// TIA Portal V20 export
// export: Created 2025-12-01T14:56:44.3017244Z, ExportSetting None, DisplayName Totally Integrated Automation Portal, DisplayVersion V20 Update 3, DisplayName TIA Portal Openness, DisplayVersion V20 Update 3, DisplayName TIA Portal Version Control Interface, DisplayVersion V20 Update 3, DisplayName STEP 7 Professional, DisplayVersion V20 Update 3, DisplayName STEP 7 Safety, DisplayVersion V20 Update 2, DisplayName WinCC Basic/Comfort/Advanced, DisplayVersion V20 Update 3, DisplayName WinCC Professional, DisplayVersion V20 Update 3, DisplayName WinCC Unified, DisplayVersion V20 Update 3
FUNCTION_BLOCK "FB246_M_STV_Carga_E1_S4"   // FB246, LAD
TITLE = Control del Ramal de Salidas
{ S7_Optimized_Access := 'FALSE' }
AUTHOR : VTD
NAME : 20160509
VERSION : 3.4
// stored: AutoNumber false, SetENOAutomatically false
   VAR_INPUT
      Mesa : UInt;   // Mesa de la FB
      Error_Tx : Bool;   // Error en el Tx
      EnTension : Bool;   // Existe Tension en la Mesa
      Termico_Tx : Bool;   // Proteccion del Tx E1E3
      pHsMx : Bool;   // pHs de la Mesa
      pHsMx_PR1 : Bool;   // pHs de Protrusion de la Mesa. Nota: No existe >> ON
      pHsMx_PR4 : Bool;   // pHs de Protrusion de la Mesa. Nota: No existe >> ON
      Avance_Tx : Bool;   // Avance del Tx
      Termico_TRx : Bool;   // Proteccion del TRx E2E4
      Pos_E2E4 : Bool;   // Pos. TR en E2E4
      Pos_E1E3 : Bool;   // Pos. TR en E1E3
      Avance_TRx : Bool;   // Avance del TRx E2E4
      EnMovimiento_TRx : Bool;   // En Movimiento la Elevacion del TRx
      LoadArrival : Bool;   // Load Arrival >>> VTD
      LoadComplete : Bool;   // LoadComplete >>> VTD
      MAnt_DescargaAct : Bool;   // E1 >> Mesa Anterior DescargaAct
      AVTF_MAnt_Mx : Bool;   // E1 >> Mesa Anterior AVTF
      P_Mens_Mant_Mx : Bool;   // E1 >> Mesa Anterior P_Mens
      PermisoPos_E2E4 : Bool;   // Permiso Pos. TR en E2E4
      PermisoPos_E1E3 : Bool;   // Permiso Pos. TR en E1E3
      Mx_PosReposo_E2E4 : Bool;   // Config >> Pos de Reposo Cargada
      Mx_TRElectrico : Bool;   // Config >> TR es Electrico
      Mx_TR_UP_E1E3 : Bool;   // Config >> TR Arriba en E1E3
      Mx_VelocidadLenta_In : Bool;   // Forzar a Velociada Lenta
      F_EnvMens_Mx : Bool;   // Fin de Envio de Mensaje
      OrdSal_S00 : Bool;   // Orden de Salida hacia el VTD
      V_CNT_pHsMx : Int := 1000;   // Valor de Presencia
      V_CNT_pHsMx_FTF : Int := 200;   // Valor para activar FTF. Nota: < = V_CNT_pHsMx.
      V_CNTSeg_pHsMx : Int := 2000;   // Valor de Seguriadad para Presencia
      V_CNT_PasoLenta : Int := 2000;   // Valor de Paso a Lenta
      V_CNT_ApHsMx : Int := 200;   // Valor de Ausencia
      V_CNTSeg_ApHsMx : Int := 2000;   // Valor de Seguriadad para Ausencia
      V_TOut_Tx_Mx : Int := 15000;   // TimeOut de Entrada por E1
      V_TOut_TR : Int := 5000;   // TimeOut de Elevacion del TR
      V_TOut_Interlock : Int := 5000;   // TimeOut de Fin del Interlock con el VTD
      V_TMP_Protrusion : Int := 200;   // TMP de Protrusion
      V_CNT_PerdidapHs : Int := 1000;   // CNT de Perdida de pHs
   END_VAR
   VAR_OUTPUT
      P_EnvMens_PMx : Bool;   // Permiso de Enviar Mensaje de Presencia
      P_EnvMens_AMx : Bool;   // Permiso de Enviar Mensaje de Ausencia
      P_RecepOK_Mx : Bool;   // Recepcion OK
      PTF_MAnt_Mx : Bool;   // E1 >> Mesa Anterior PTF
      FTF_MAnt_Mx : Bool;   // E1 >> Mesa Anterior FTF
   END_VAR
   VAR
      Anular_prE1 : Bool;   // ???
      Anular_prS4 : Bool;   // ???
      Mx_ET00 : Bool;
      Mx_ET01 : Bool;
      Mx_ET02 : Bool;
      Mx_ET08 : Bool;
      Mx_ET09 : Bool;
      Mx_ET10 : Bool;
      Mx_ET11 : Bool;
      Mx_ET12 : Bool;
      Mx_ET110 : Bool;
      Mx_ET111 : Bool;
      Mx_ET50 : Bool;
      Mx_ET51 : Bool;
      Mx_ET52 : Bool;
      Mx_ET150 : Bool;
      Mx_ET151 : Bool;
      Mx_ET152 : Bool;
      ProtocoloIniciado : Bool;   // Iniciado el Envio del Mensaje de Presencia
      CNT_pHsMx_FTF_OK : Bool;   // Enviar ya FTF
      STAT_EnvMens_PMx : Bool;   // Interna >> Envio del Mensaje de Presencia
      STAT_EnvMens_AMx : Bool;   // Interna >> Envio de Mensaje de Ausencia
      STAT_FTF_MAnt_Mx : Bool;   // Interna >> FTF de MAnt >> Mx
      CNT_pHsMx { S7_SetPoint := 'True'} : "FB910_CNT_UHS";   // CNT de la Presencia
      CNTSeg_pHsMx { S7_SetPoint := 'True'} : "FB910_CNT_UHS";   // CNT de Seguridad de la Presencia
      CNT_ApHsMx { S7_SetPoint := 'True'} : "FB910_CNT_UHS";   // CNT de la Ausencia
      CNTSeg_ApHsMx { S7_SetPoint := 'True'} : "FB910_CNT_UHS";   // CNT de Seguridad de la Ausencia
      TMP_EnTension { S7_SetPoint := 'True'} : "FB910_CNT_UHS";
      TOut_Av_Mx { S7_SetPoint := 'True'} : "FB910_CNT_UHS";   // Time Out de Entrada de E1
      TOut_Subir_TR { S7_SetPoint := 'True'} : "FB910_CNT_UHS";   // Time Out de Subida del TR
      TOut_Bajar_TR { S7_SetPoint := 'True'} : "FB910_CNT_UHS";   // Time Out de Bajada del TR
      TOut_Interlock { S7_SetPoint := 'True'} : "FB910_CNT_UHS";   // Time Out de Fin de Interlock con el VTD
      TMP_Protrusion { S7_SetPoint := 'True'} : "FB910_CNT_UHS";   // TMP de la Protrusion
      CNT_PerdidapHs { S7_SetPoint := 'True'} : "FB910_CNT_UHS";   // CNT de Perdida de pHs
      Interlock_manual { S7_SetPoint := 'True'} : "UDT_Interlock_manual_STV";
   END_VAR
   VAR_TEMP
      EstadoZona : "EstadoZona";   // Estado de Zona de la Mesa
      EstadoVI : "EstadosMesa";   // Estado del Vehiculo Inteliguente de la Mesa
      ConfigFB : "UDT_ConfigFB";   // Configuracion de la FB de la Mesa
      Interlock : "UDT_Interlock_STV";
      V_Protrusion : Int;
      retval : Int;
      cero : USInt;
      Aux_ET00 : Bool;
   END_VAR
BEGIN

REGION Network 1: INICIALIZAR - Recoger las Variables de Estado de la Mesa
   // Se recoge - Estado_CBx
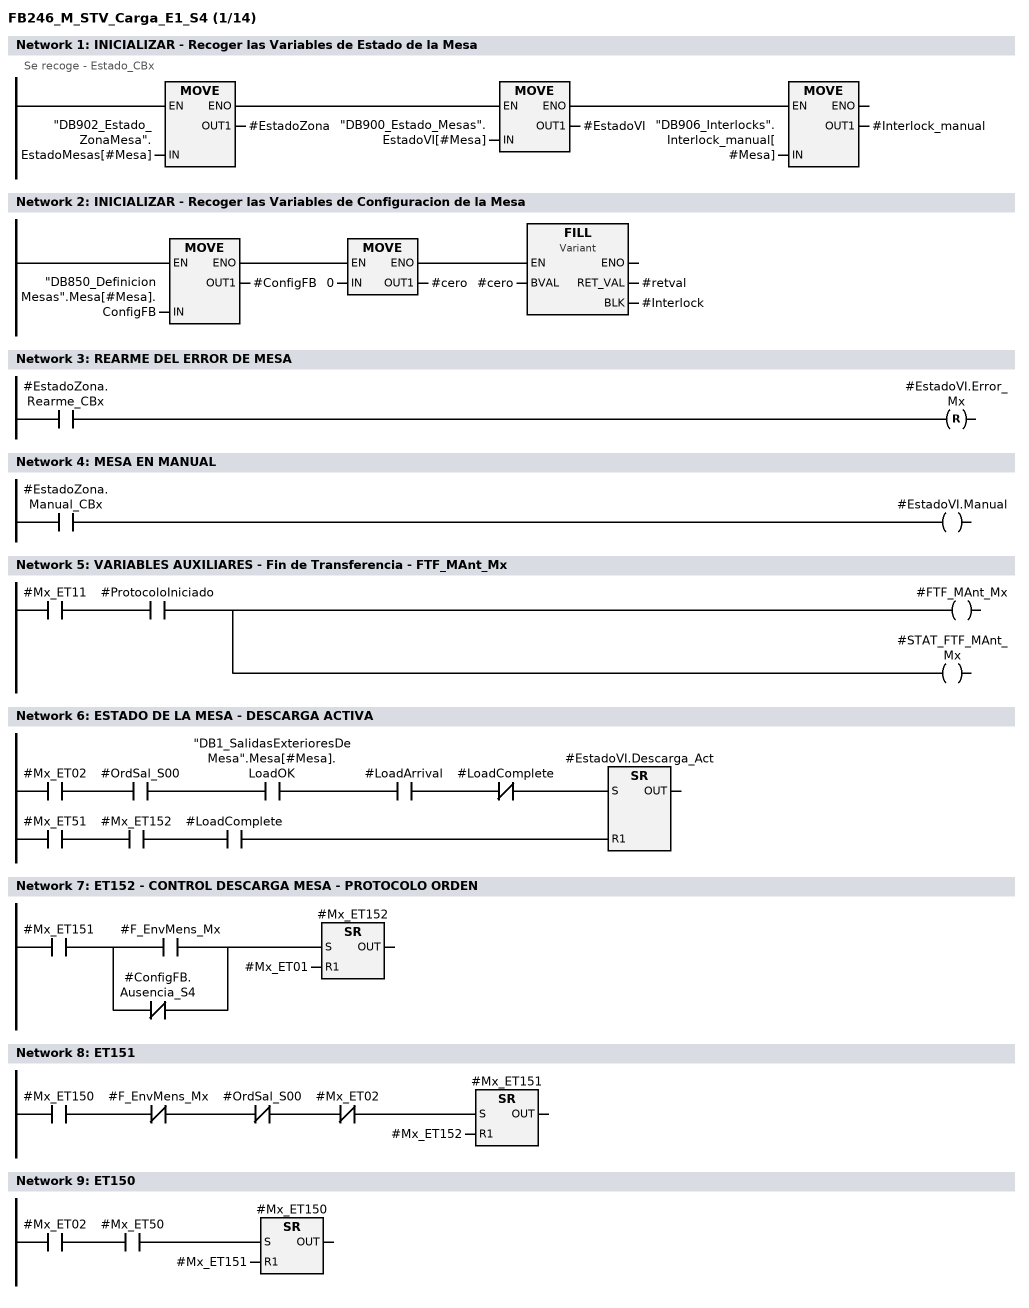
   RUNG wire#powerrail
      Move(in := "DB902_Estado_ZonaMesa".EstadoMesas[#Mesa], out1 => #EstadoZona)
      Move(in := "DB900_Estado_Mesas".EstadoVI[#Mesa], out1 => #EstadoVI)
      Move(in := "DB906_Interlocks".Interlock_manual[#Mesa], out1 => #Interlock_manual)
   END_RUNG
   // the same network as SCL:
   #EstadoZona := "DB902_Estado_ZonaMesa".EstadoMesas[#Mesa];
   #EstadoVI := "DB900_Estado_Mesas".EstadoVI[#Mesa];
   #Interlock_manual := "DB906_Interlocks".Interlock_manual[#Mesa];
END_REGION

REGION Network 2: INICIALIZAR - Recoger las Variables de Configuracion de la Mesa
   RUNG wire#powerrail
      Move(in := "DB850_DefinicionMesas".Mesa[#Mesa].ConfigFB, out1 => #ConfigFB)
      Move(in := 0, out1 => #cero)
      { S7_Templates := "ptr_type := Variant" } FILL(BVAL := #cero, RET_VAL => #retval, BLK => #Interlock)
   END_RUNG
   // the same network as SCL:
   #ConfigFB := "DB850_DefinicionMesas".Mesa[#Mesa].ConfigFB;
   #cero := 0;
   #retval := FILL(BVAL := #cero, BLK => #Interlock);
END_REGION

REGION Network 3: REARME DEL ERROR DE MESA
   RUNG wire#powerrail
      Contact( #EstadoZona.Rearme_CBx )
      R_Coil( #EstadoVI.Error_Mx )
   END_RUNG
   // the same network as SCL:
   IF #EstadoZona.Rearme_CBx THEN #EstadoVI.Error_Mx := FALSE; END_IF;
END_REGION

REGION Network 4: MESA EN MANUAL
   RUNG wire#powerrail
      Contact( #EstadoZona.Manual_CBx )
      Coil( #EstadoVI.Manual )
   END_RUNG
   // the same network as SCL:
   #EstadoVI.Manual := #EstadoZona.Manual_CBx;
END_REGION

REGION Network 5: VARIABLES AUXILIARES - Fin de Transferencia - FTF_MAnt_Mx
   RUNG wire#powerrail
      Contact( #Mx_ET11 )
      Contact( #ProtocoloIniciado )
      wire#w1
      Coil( #FTF_MAnt_Mx )
   END_RUNG
   RUNG wire#w1
      Coil( #STAT_FTF_MAnt_Mx )
   END_RUNG
   // the same network as SCL:
   #FTF_MAnt_Mx := #Mx_ET11 AND #ProtocoloIniciado;
   #STAT_FTF_MAnt_Mx := #FTF_MAnt_Mx;
END_REGION

REGION Network 6: ESTADO DE LA MESA - DESCARGA ACTIVA
   RUNG wire#powerrail
      Contact( #Mx_ET02 )
      Contact( #OrdSal_S00 )
      Contact( "DB1_SalidasExterioresDeMesa".Mesa[#Mesa].LoadOK )
      Contact( #LoadArrival )
      I_Contact( #LoadComplete )
      S_SR(operand := #EstadoVI.Descarga_Act, r1 := wire#w1)
   END_RUNG
   RUNG wire#powerrail
      Contact( #Mx_ET51 )
      Contact( #Mx_ET152 )
      Contact( #LoadComplete )
   END_RUNG wire#w1
   // the same network as SCL:
   IF #Mx_ET02 AND #OrdSal_S00 AND "DB1_SalidasExterioresDeMesa".Mesa[#Mesa].LoadOK AND #LoadArrival AND NOT #LoadComplete THEN
       #EstadoVI.Descarga_Act := TRUE;   // SR flip-flop
   END_IF;
   IF #Mx_ET51 AND #Mx_ET152 AND #LoadComplete THEN #EstadoVI.Descarga_Act := FALSE; END_IF;
END_REGION

REGION Network 7: ET152 - CONTROL DESCARGA MESA - PROTOCOLO ORDEN
   RUNG wire#powerrail
      Contact( #Mx_ET151 )
      wire#w1
      Contact( #F_EnvMens_Mx )
      wire#w2
      S_SR(operand := #Mx_ET152, r1 := #Mx_ET01)
   END_RUNG
   RUNG wire#w1
      I_Contact( #ConfigFB.Ausencia_S4 )
   END_RUNG wire#w2
   // the same network as SCL:
   IF #Mx_ET151 AND (#F_EnvMens_Mx OR NOT #ConfigFB.Ausencia_S4) THEN
       #Mx_ET152 := TRUE;   // SR flip-flop
   END_IF;
   IF #Mx_ET01 THEN #Mx_ET152 := FALSE; END_IF;
END_REGION

REGION Network 8: ET151
   RUNG wire#powerrail
      Contact( #Mx_ET150 )
      I_Contact( #F_EnvMens_Mx )
      I_Contact( #OrdSal_S00 )
      I_Contact( #Mx_ET02 )
      S_SR(operand := #Mx_ET151, r1 := #Mx_ET152)
   END_RUNG
   // the same network as SCL:
   IF #Mx_ET150 AND NOT #F_EnvMens_Mx AND NOT #OrdSal_S00 AND NOT #Mx_ET02 THEN
       #Mx_ET151 := TRUE;   // SR flip-flop
   END_IF;
   IF #Mx_ET152 THEN #Mx_ET151 := FALSE; END_IF;
END_REGION

REGION Network 9: ET150
   RUNG wire#powerrail
      Contact( #Mx_ET02 )
      Contact( #Mx_ET50 )
      S_SR(operand := #Mx_ET150, r1 := #Mx_ET151)
   END_RUNG
   // the same network as SCL:
   IF #Mx_ET02 AND #Mx_ET50 THEN
       #Mx_ET150 := TRUE;   // SR flip-flop
   END_IF;
   IF #Mx_ET151 THEN #Mx_ET150 := FALSE; END_IF;
END_REGION

REGION Network 10: ET52 - CONTROL DESCARGA MESA
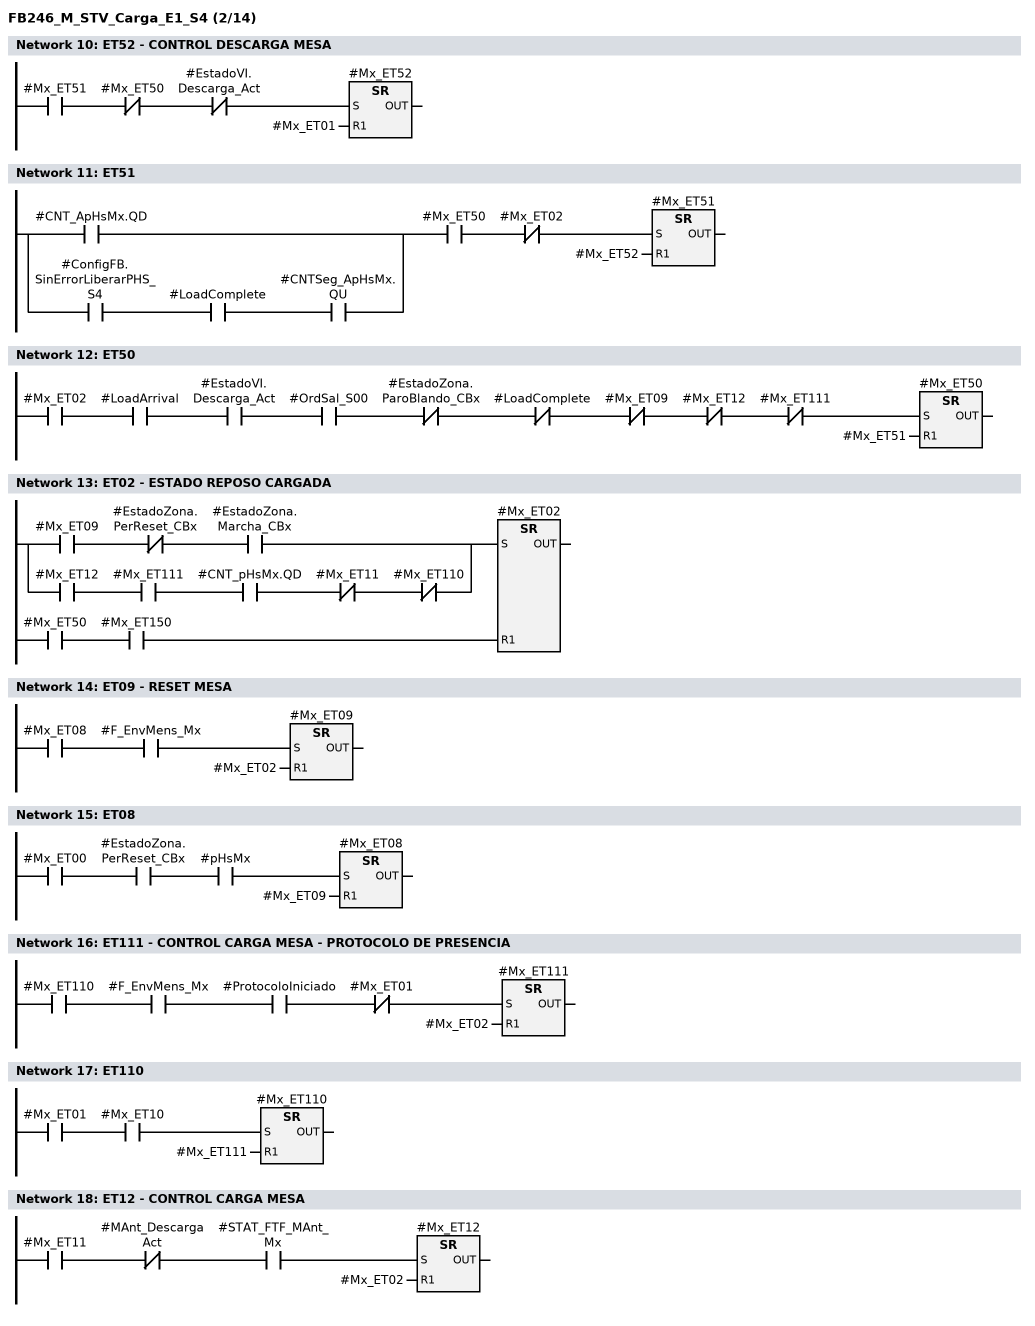
   RUNG wire#powerrail
      Contact( #Mx_ET51 )
      I_Contact( #Mx_ET50 )
      I_Contact( #EstadoVI.Descarga_Act )
      S_SR(operand := #Mx_ET52, r1 := #Mx_ET01)
   END_RUNG
   // the same network as SCL:
   IF #Mx_ET51 AND NOT #Mx_ET50 AND NOT #EstadoVI.Descarga_Act THEN
       #Mx_ET52 := TRUE;   // SR flip-flop
   END_IF;
   IF #Mx_ET01 THEN #Mx_ET52 := FALSE; END_IF;
END_REGION

REGION Network 11: ET51
   RUNG wire#powerrail
      Contact( #CNT_ApHsMx.QD )
      wire#w1
      Contact( #Mx_ET50 )
      I_Contact( #Mx_ET02 )
      S_SR(operand := #Mx_ET51, r1 := #Mx_ET52)
   END_RUNG
   RUNG wire#powerrail
      Contact( #ConfigFB.SinErrorLiberarPHS_S4 )
      Contact( #LoadComplete )
      Contact( #CNTSeg_ApHsMx.QU )
   END_RUNG wire#w1
   // the same network as SCL:
   IF (#CNT_ApHsMx.QD OR (#ConfigFB.SinErrorLiberarPHS_S4 AND #LoadComplete AND #CNTSeg_ApHsMx.QU)) AND #Mx_ET50 AND NOT #Mx_ET02 THEN
       #Mx_ET51 := TRUE;   // SR flip-flop
   END_IF;
   IF #Mx_ET52 THEN #Mx_ET51 := FALSE; END_IF;
END_REGION

REGION Network 12: ET50
   RUNG wire#powerrail
      Contact( #Mx_ET02 )
      Contact( #LoadArrival )
      Contact( #EstadoVI.Descarga_Act )
      Contact( #OrdSal_S00 )
      I_Contact( #EstadoZona.ParoBlando_CBx )
      I_Contact( #LoadComplete )
      I_Contact( #Mx_ET09 )
      I_Contact( #Mx_ET12 )
      I_Contact( #Mx_ET111 )
      S_SR(operand := #Mx_ET50, r1 := #Mx_ET51)
   END_RUNG
   // the same network as SCL:
   IF #Mx_ET02 AND #LoadArrival AND #EstadoVI.Descarga_Act AND #OrdSal_S00 AND NOT #EstadoZona.ParoBlando_CBx AND NOT #LoadComplete AND NOT #Mx_ET09 AND NOT #Mx_ET12 AND NOT #Mx_ET111 THEN
       #Mx_ET50 := TRUE;   // SR flip-flop
   END_IF;
   IF #Mx_ET51 THEN #Mx_ET50 := FALSE; END_IF;
END_REGION

REGION Network 13: ET02 - ESTADO REPOSO CARGADA
   RUNG wire#powerrail
      Contact( #Mx_ET09 )
      I_Contact( #EstadoZona.PerReset_CBx )
      Contact( #EstadoZona.Marcha_CBx )
      wire#w1
      S_SR(operand := #Mx_ET02, r1 := wire#w2)
   END_RUNG
   RUNG wire#powerrail
      Contact( #Mx_ET12 )
      Contact( #Mx_ET111 )
      Contact( #CNT_pHsMx.QD )
      I_Contact( #Mx_ET11 )
      I_Contact( #Mx_ET110 )
   END_RUNG wire#w1
   RUNG wire#powerrail
      Contact( #Mx_ET50 )
      Contact( #Mx_ET150 )
   END_RUNG wire#w2
   // the same network as SCL:
   IF (#Mx_ET09 AND NOT #EstadoZona.PerReset_CBx AND #EstadoZona.Marcha_CBx) OR (#Mx_ET12 AND #Mx_ET111 AND #CNT_pHsMx.QD AND NOT #Mx_ET11 AND NOT #Mx_ET110) THEN
       #Mx_ET02 := TRUE;   // SR flip-flop
   END_IF;
   IF #Mx_ET50 AND #Mx_ET150 THEN #Mx_ET02 := FALSE; END_IF;
END_REGION

REGION Network 14: ET09 - RESET MESA
   RUNG wire#powerrail
      Contact( #Mx_ET08 )
      Contact( #F_EnvMens_Mx )
      S_SR(operand := #Mx_ET09, r1 := #Mx_ET02)
   END_RUNG
   // the same network as SCL:
   IF #Mx_ET08 AND #F_EnvMens_Mx THEN
       #Mx_ET09 := TRUE;   // SR flip-flop
   END_IF;
   IF #Mx_ET02 THEN #Mx_ET09 := FALSE; END_IF;
END_REGION

REGION Network 15: ET08
   RUNG wire#powerrail
      Contact( #Mx_ET00 )
      Contact( #EstadoZona.PerReset_CBx )
      Contact( #pHsMx )
      S_SR(operand := #Mx_ET08, r1 := #Mx_ET09)
   END_RUNG
   // the same network as SCL:
   IF #Mx_ET00 AND #EstadoZona.PerReset_CBx AND #pHsMx THEN
       #Mx_ET08 := TRUE;   // SR flip-flop
   END_IF;
   IF #Mx_ET09 THEN #Mx_ET08 := FALSE; END_IF;
END_REGION

REGION Network 16: ET111 - CONTROL CARGA MESA - PROTOCOLO DE PRESENCIA
   RUNG wire#powerrail
      Contact( #Mx_ET110 )
      Contact( #F_EnvMens_Mx )
      Contact( #ProtocoloIniciado )
      I_Contact( #Mx_ET01 )
      S_SR(operand := #Mx_ET111, r1 := #Mx_ET02)
   END_RUNG
   // the same network as SCL:
   IF #Mx_ET110 AND #F_EnvMens_Mx AND #ProtocoloIniciado AND NOT #Mx_ET01 THEN
       #Mx_ET111 := TRUE;   // SR flip-flop
   END_IF;
   IF #Mx_ET02 THEN #Mx_ET111 := FALSE; END_IF;
END_REGION

REGION Network 17: ET110
   RUNG wire#powerrail
      Contact( #Mx_ET01 )
      Contact( #Mx_ET10 )
      S_SR(operand := #Mx_ET110, r1 := #Mx_ET111)
   END_RUNG
   // the same network as SCL:
   IF #Mx_ET01 AND #Mx_ET10 THEN
       #Mx_ET110 := TRUE;   // SR flip-flop
   END_IF;
   IF #Mx_ET111 THEN #Mx_ET110 := FALSE; END_IF;
END_REGION

REGION Network 18: ET12 - CONTROL CARGA MESA
   RUNG wire#powerrail
      Contact( #Mx_ET11 )
      I_Contact( #MAnt_DescargaAct )
      Contact( #STAT_FTF_MAnt_Mx )
      S_SR(operand := #Mx_ET12, r1 := #Mx_ET02)
   END_RUNG
   // the same network as SCL:
   IF #Mx_ET11 AND NOT #MAnt_DescargaAct AND #STAT_FTF_MAnt_Mx THEN
       #Mx_ET12 := TRUE;   // SR flip-flop
   END_IF;
   IF #Mx_ET02 THEN #Mx_ET12 := FALSE; END_IF;
END_REGION

REGION Network 19: ET11
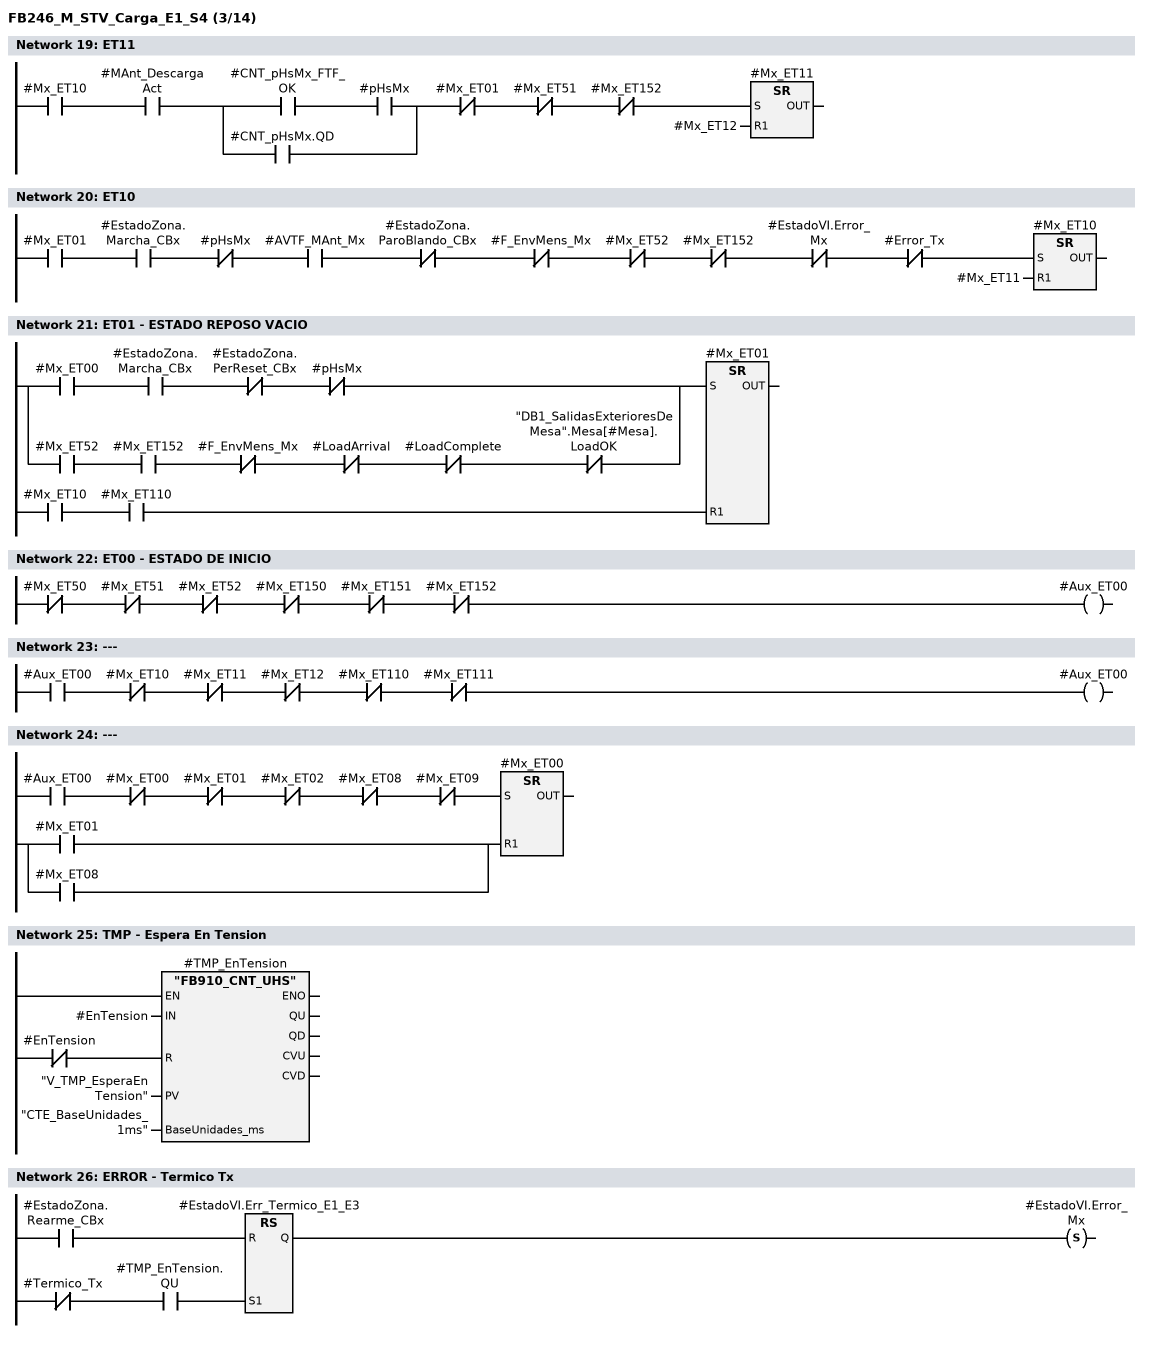
   RUNG wire#powerrail
      Contact( #Mx_ET10 )
      Contact( #MAnt_DescargaAct )
      wire#w1
      Contact( #CNT_pHsMx_FTF_OK )
      Contact( #pHsMx )
      wire#w2
      I_Contact( #Mx_ET01 )
      I_Contact( #Mx_ET51 )
      I_Contact( #Mx_ET152 )
      S_SR(operand := #Mx_ET11, r1 := #Mx_ET12)
   END_RUNG
   RUNG wire#w1
      Contact( #CNT_pHsMx.QD )
   END_RUNG wire#w2
   // the same network as SCL:
   IF #Mx_ET10 AND #MAnt_DescargaAct AND ((#CNT_pHsMx_FTF_OK AND #pHsMx) OR #CNT_pHsMx.QD) AND NOT #Mx_ET01 AND NOT #Mx_ET51 AND NOT #Mx_ET152 THEN
       #Mx_ET11 := TRUE;   // SR flip-flop
   END_IF;
   IF #Mx_ET12 THEN #Mx_ET11 := FALSE; END_IF;
END_REGION

REGION Network 20: ET10
   RUNG wire#powerrail
      Contact( #Mx_ET01 )
      Contact( #EstadoZona.Marcha_CBx )
      I_Contact( #pHsMx )
      Contact( #AVTF_MAnt_Mx )
      I_Contact( #EstadoZona.ParoBlando_CBx )
      I_Contact( #F_EnvMens_Mx )
      I_Contact( #Mx_ET52 )
      I_Contact( #Mx_ET152 )
      I_Contact( #EstadoVI.Error_Mx )
      I_Contact( #Error_Tx )
      S_SR(operand := #Mx_ET10, r1 := #Mx_ET11)
   END_RUNG
   // the same network as SCL:
   IF #Mx_ET01 AND #EstadoZona.Marcha_CBx AND NOT #pHsMx AND #AVTF_MAnt_Mx AND NOT #EstadoZona.ParoBlando_CBx AND NOT #F_EnvMens_Mx AND NOT #Mx_ET52 AND NOT #Mx_ET152 AND NOT #EstadoVI.Error_Mx AND NOT #Error_Tx THEN
       #Mx_ET10 := TRUE;   // SR flip-flop
   END_IF;
   IF #Mx_ET11 THEN #Mx_ET10 := FALSE; END_IF;
END_REGION

REGION Network 21: ET01 - ESTADO REPOSO VACIO
   RUNG wire#powerrail
      Contact( #Mx_ET00 )
      Contact( #EstadoZona.Marcha_CBx )
      I_Contact( #EstadoZona.PerReset_CBx )
      I_Contact( #pHsMx )
      wire#w1
      S_SR(operand := #Mx_ET01, r1 := wire#w2)
   END_RUNG
   RUNG wire#powerrail
      Contact( #Mx_ET52 )
      Contact( #Mx_ET152 )
      I_Contact( #F_EnvMens_Mx )
      I_Contact( #LoadArrival )
      I_Contact( #LoadComplete )
      I_Contact( "DB1_SalidasExterioresDeMesa".Mesa[#Mesa].LoadOK )
   END_RUNG wire#w1
   RUNG wire#powerrail
      Contact( #Mx_ET10 )
      Contact( #Mx_ET110 )
   END_RUNG wire#w2
   // the same network as SCL:
   IF (#Mx_ET00 AND #EstadoZona.Marcha_CBx AND NOT #EstadoZona.PerReset_CBx AND NOT #pHsMx) OR (#Mx_ET52 AND #Mx_ET152 AND NOT #F_EnvMens_Mx AND NOT #LoadArrival AND NOT #LoadComplete AND NOT "DB1_SalidasExterioresDeMesa".Mesa[#Mesa].LoadOK) THEN
       #Mx_ET01 := TRUE;   // SR flip-flop
   END_IF;
   IF #Mx_ET10 AND #Mx_ET110 THEN #Mx_ET01 := FALSE; END_IF;
END_REGION

REGION Network 22: ET00 - ESTADO DE INICIO
   RUNG wire#powerrail
      I_Contact( #Mx_ET50 )
      I_Contact( #Mx_ET51 )
      I_Contact( #Mx_ET52 )
      I_Contact( #Mx_ET150 )
      I_Contact( #Mx_ET151 )
      I_Contact( #Mx_ET152 )
      Coil( #Aux_ET00 )
   END_RUNG
   // the same network as SCL:
   #Aux_ET00 := NOT #Mx_ET50 AND NOT #Mx_ET51 AND NOT #Mx_ET52 AND NOT #Mx_ET150 AND NOT #Mx_ET151 AND NOT #Mx_ET152;
END_REGION

REGION Network 23: ---
   RUNG wire#powerrail
      Contact( #Aux_ET00 )
      I_Contact( #Mx_ET10 )
      I_Contact( #Mx_ET11 )
      I_Contact( #Mx_ET12 )
      I_Contact( #Mx_ET110 )
      I_Contact( #Mx_ET111 )
      Coil( #Aux_ET00 )
   END_RUNG
   // the same network as SCL:
   #Aux_ET00 := #Aux_ET00 AND NOT #Mx_ET10 AND NOT #Mx_ET11 AND NOT #Mx_ET12 AND NOT #Mx_ET110 AND NOT #Mx_ET111;
END_REGION

REGION Network 24: ---
   RUNG wire#powerrail
      Contact( #Aux_ET00 )
      I_Contact( #Mx_ET00 )
      I_Contact( #Mx_ET01 )
      I_Contact( #Mx_ET02 )
      I_Contact( #Mx_ET08 )
      I_Contact( #Mx_ET09 )
      S_SR(operand := #Mx_ET00, r1 := wire#w1)
   END_RUNG
   RUNG wire#powerrail
      Contact( #Mx_ET01 )
   END_RUNG wire#w1
   RUNG wire#powerrail
      Contact( #Mx_ET08 )
   END_RUNG wire#w1
   // the same network as SCL:
   IF #Aux_ET00 AND NOT #Mx_ET00 AND NOT #Mx_ET01 AND NOT #Mx_ET02 AND NOT #Mx_ET08 AND NOT #Mx_ET09 THEN
       #Mx_ET00 := TRUE;   // SR flip-flop
   END_IF;
   IF #Mx_ET01 OR #Mx_ET08 THEN #Mx_ET00 := FALSE; END_IF;
END_REGION

REGION Network 25: TMP - Espera En Tension
   RUNG wire#powerrail
      #TMP_EnTension(R := wire#w1, IN := #EnTension, PV := "V_TMP_EsperaEnTension", BaseUnidades_ms := "CTE_BaseUnidades_1ms", QU =>, QD =>, CVU =>, CVD =>)
   END_RUNG
   RUNG wire#powerrail
      I_Contact( #EnTension )
   END_RUNG wire#w1
   // the same network as SCL:
   #TMP_EnTension(IN := #EnTension,   // "FB910_CNT_UHS"
                  R := NOT #EnTension,
                  PV := "V_TMP_EsperaEnTension",
                  BaseUnidades_ms := "CTE_BaseUnidades_1ms");
END_REGION

REGION Network 26: ERROR - Termico Tx
   RUNG wire#powerrail
      Contact( #EstadoZona.Rearme_CBx )
      S_RS(operand := #EstadoVI.Err_Termico_E1_E3, s1 := wire#w1)
      S_Coil( #EstadoVI.Error_Mx )
   END_RUNG
   RUNG wire#powerrail
      I_Contact( #Termico_Tx )
      Contact( #TMP_EnTension.QU )
   END_RUNG wire#w1
   // the same network as SCL:
   IF #EstadoZona.Rearme_CBx THEN
       #EstadoVI.Err_Termico_E1_E3 := FALSE;   // RS flip-flop
   END_IF;
   IF NOT #Termico_Tx AND #TMP_EnTension.QU THEN #EstadoVI.Err_Termico_E1_E3 := TRUE; END_IF;
   IF #EstadoVI.Err_Termico_E1_E3 THEN #EstadoVI.Error_Mx := TRUE; END_IF;
END_REGION

REGION Network 27: ERROR - Termico TRx
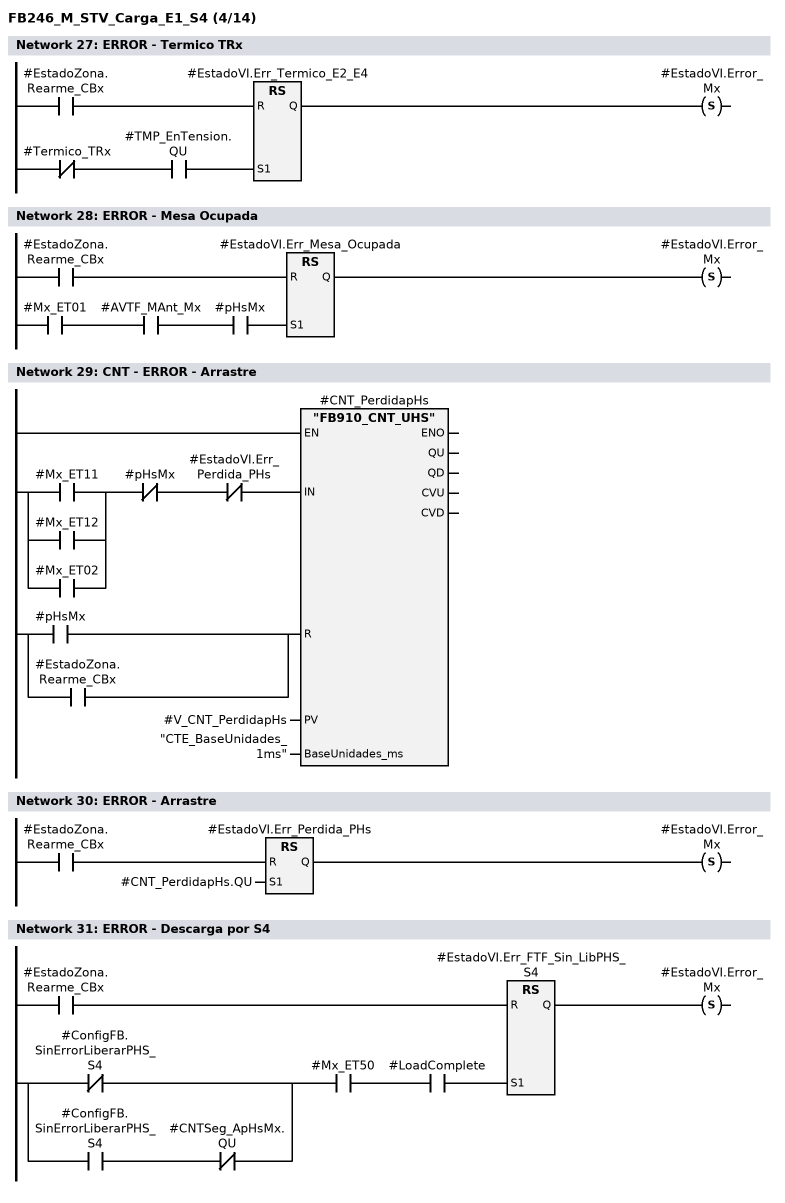
   RUNG wire#powerrail
      Contact( #EstadoZona.Rearme_CBx )
      S_RS(operand := #EstadoVI.Err_Termico_E2_E4, s1 := wire#w1)
      S_Coil( #EstadoVI.Error_Mx )
   END_RUNG
   RUNG wire#powerrail
      I_Contact( #Termico_TRx )
      Contact( #TMP_EnTension.QU )
   END_RUNG wire#w1
   // the same network as SCL:
   IF #EstadoZona.Rearme_CBx THEN
       #EstadoVI.Err_Termico_E2_E4 := FALSE;   // RS flip-flop
   END_IF;
   IF NOT #Termico_TRx AND #TMP_EnTension.QU THEN #EstadoVI.Err_Termico_E2_E4 := TRUE; END_IF;
   IF #EstadoVI.Err_Termico_E2_E4 THEN #EstadoVI.Error_Mx := TRUE; END_IF;
END_REGION

REGION Network 28: ERROR - Mesa Ocupada
   RUNG wire#powerrail
      Contact( #EstadoZona.Rearme_CBx )
      S_RS(operand := #EstadoVI.Err_Mesa_Ocupada, s1 := wire#w1)
      S_Coil( #EstadoVI.Error_Mx )
   END_RUNG
   RUNG wire#powerrail
      Contact( #Mx_ET01 )
      Contact( #AVTF_MAnt_Mx )
      Contact( #pHsMx )
   END_RUNG wire#w1
   // the same network as SCL:
   IF #EstadoZona.Rearme_CBx THEN
       #EstadoVI.Err_Mesa_Ocupada := FALSE;   // RS flip-flop
   END_IF;
   IF #Mx_ET01 AND #AVTF_MAnt_Mx AND #pHsMx THEN #EstadoVI.Err_Mesa_Ocupada := TRUE; END_IF;
   IF #EstadoVI.Err_Mesa_Ocupada THEN #EstadoVI.Error_Mx := TRUE; END_IF;
END_REGION

REGION Network 29: CNT - ERROR - Arrastre
   RUNG wire#powerrail
      #CNT_PerdidapHs(IN := wire#w2, R := wire#w3, PV := #V_CNT_PerdidapHs, BaseUnidades_ms := "CTE_BaseUnidades_1ms", QU =>, QD =>, CVU =>, CVD =>)
   END_RUNG
   RUNG wire#powerrail
      Contact( #Mx_ET11 )
      wire#w1
      I_Contact( #pHsMx )
      I_Contact( #EstadoVI.Err_Perdida_PHs )
   END_RUNG wire#w2
   RUNG wire#powerrail
      Contact( #Mx_ET12 )
   END_RUNG wire#w1
   RUNG wire#powerrail
      Contact( #Mx_ET02 )
   END_RUNG wire#w1
   RUNG wire#powerrail
      Contact( #pHsMx )
   END_RUNG wire#w3
   RUNG wire#powerrail
      Contact( #EstadoZona.Rearme_CBx )
   END_RUNG wire#w3
   // the same network as SCL:
   #CNT_PerdidapHs(IN := (#Mx_ET11 OR #Mx_ET12 OR #Mx_ET02) AND NOT #pHsMx AND NOT #EstadoVI.Err_Perdida_PHs,   // "FB910_CNT_UHS"
                   R := #pHsMx OR #EstadoZona.Rearme_CBx,
                   PV := #V_CNT_PerdidapHs,
                   BaseUnidades_ms := "CTE_BaseUnidades_1ms");
END_REGION

REGION Network 30: ERROR - Arrastre
   RUNG wire#powerrail
      Contact( #EstadoZona.Rearme_CBx )
      S_RS(operand := #EstadoVI.Err_Perdida_PHs, s1 := #CNT_PerdidapHs.QU)
      S_Coil( #EstadoVI.Error_Mx )
   END_RUNG
   // the same network as SCL:
   IF #EstadoZona.Rearme_CBx THEN
       #EstadoVI.Err_Perdida_PHs := FALSE;   // RS flip-flop
   END_IF;
   IF #CNT_PerdidapHs.QU THEN #EstadoVI.Err_Perdida_PHs := TRUE; END_IF;
   IF #EstadoVI.Err_Perdida_PHs THEN #EstadoVI.Error_Mx := TRUE; END_IF;
END_REGION

REGION Network 31: ERROR - Descarga por S4
   RUNG wire#powerrail
      Contact( #EstadoZona.Rearme_CBx )
      S_RS(operand := #EstadoVI.Err_FTF_Sin_LibPHS_S4, s1 := wire#w2)
      S_Coil( #EstadoVI.Error_Mx )
   END_RUNG
   RUNG wire#powerrail
      I_Contact( #ConfigFB.SinErrorLiberarPHS_S4 )
      wire#w1
      Contact( #Mx_ET50 )
      Contact( #LoadComplete )
   END_RUNG wire#w2
   RUNG wire#powerrail
      Contact( #ConfigFB.SinErrorLiberarPHS_S4 )
      I_Contact( #CNTSeg_ApHsMx.QU )
   END_RUNG wire#w1
   // the same network as SCL:
   IF #EstadoZona.Rearme_CBx THEN
       #EstadoVI.Err_FTF_Sin_LibPHS_S4 := FALSE;   // RS flip-flop
   END_IF;
   IF (NOT #ConfigFB.SinErrorLiberarPHS_S4 OR (#ConfigFB.SinErrorLiberarPHS_S4 AND NOT #CNTSeg_ApHsMx.QU)) AND #Mx_ET50 AND #LoadComplete THEN
       #EstadoVI.Err_FTF_Sin_LibPHS_S4 := TRUE;
   END_IF;
   IF #EstadoVI.Err_FTF_Sin_LibPHS_S4 THEN #EstadoVI.Error_Mx := TRUE; END_IF;
END_REGION

REGION Network 32: TMP - ERROR - TimeOut Avance Tx
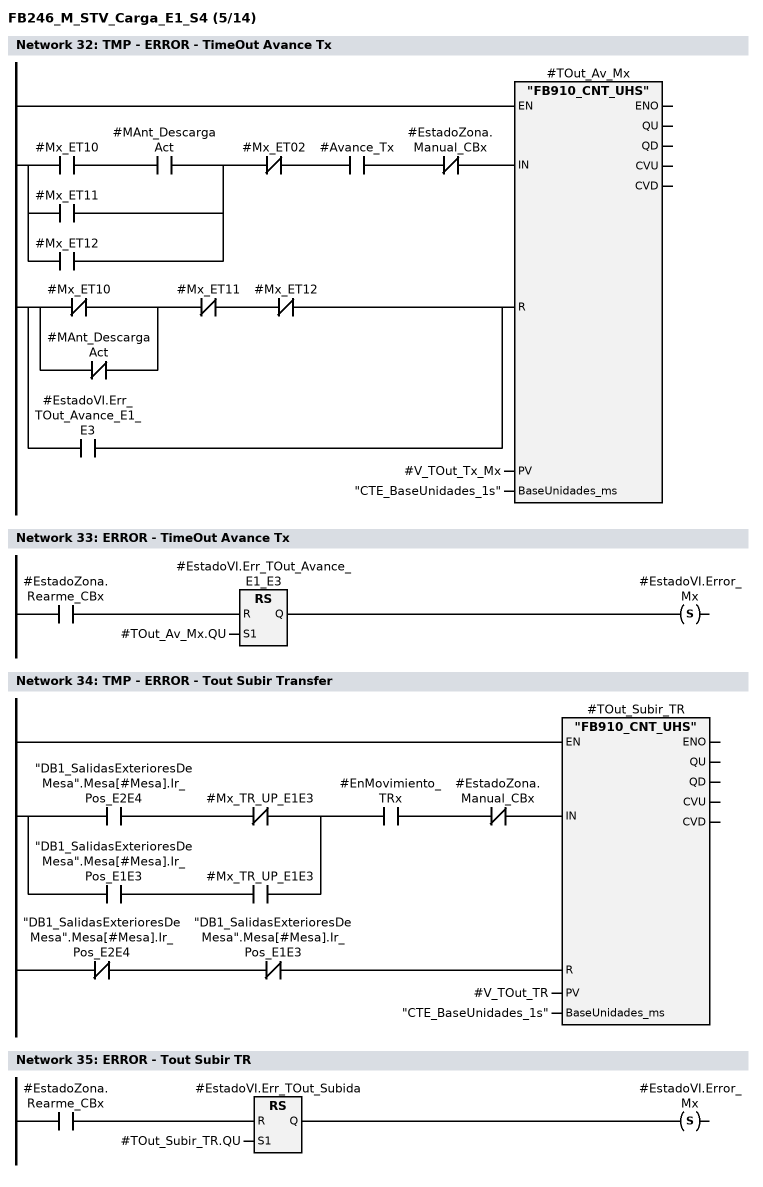
   RUNG wire#powerrail
      #TOut_Av_Mx(IN := wire#w2, R := wire#w4, PV := #V_TOut_Tx_Mx, BaseUnidades_ms := "CTE_BaseUnidades_1s", QU =>, QD =>, CVU =>, CVD =>)
   END_RUNG
   RUNG wire#powerrail
      Contact( #Mx_ET10 )
      Contact( #MAnt_DescargaAct )
      wire#w1
      I_Contact( #Mx_ET02 )
      Contact( #Avance_Tx )
      I_Contact( #EstadoZona.Manual_CBx )
   END_RUNG wire#w2
   RUNG wire#powerrail
      Contact( #Mx_ET11 )
   END_RUNG wire#w1
   RUNG wire#powerrail
      Contact( #Mx_ET12 )
   END_RUNG wire#w1
   RUNG wire#powerrail
      I_Contact( #Mx_ET10 )
      wire#w3
      I_Contact( #Mx_ET11 )
      I_Contact( #Mx_ET12 )
   END_RUNG wire#w4
   RUNG wire#powerrail
      I_Contact( #MAnt_DescargaAct )
   END_RUNG wire#w3
   RUNG wire#powerrail
      Contact( #EstadoVI.Err_TOut_Avance_E1_E3 )
   END_RUNG wire#w4
   // the same network as SCL:
   #TOut_Av_Mx(IN := ((#Mx_ET10 AND #MAnt_DescargaAct) OR #Mx_ET11 OR #Mx_ET12) AND NOT #Mx_ET02 AND #Avance_Tx AND NOT #EstadoZona.Manual_CBx,   // "FB910_CNT_UHS"
               R := ((NOT #Mx_ET10 OR NOT #MAnt_DescargaAct) AND NOT #Mx_ET11 AND NOT #Mx_ET12) OR #EstadoVI.Err_TOut_Avance_E1_E3,
               PV := #V_TOut_Tx_Mx,
               BaseUnidades_ms := "CTE_BaseUnidades_1s");
END_REGION

REGION Network 33: ERROR - TimeOut Avance Tx
   RUNG wire#powerrail
      Contact( #EstadoZona.Rearme_CBx )
      S_RS(operand := #EstadoVI.Err_TOut_Avance_E1_E3, s1 := #TOut_Av_Mx.QU)
      S_Coil( #EstadoVI.Error_Mx )
   END_RUNG
   // the same network as SCL:
   IF #EstadoZona.Rearme_CBx THEN
       #EstadoVI.Err_TOut_Avance_E1_E3 := FALSE;   // RS flip-flop
   END_IF;
   IF #TOut_Av_Mx.QU THEN #EstadoVI.Err_TOut_Avance_E1_E3 := TRUE; END_IF;
   IF #EstadoVI.Err_TOut_Avance_E1_E3 THEN #EstadoVI.Error_Mx := TRUE; END_IF;
END_REGION

REGION Network 34: TMP - ERROR - Tout Subir Transfer
   RUNG wire#powerrail
      #TOut_Subir_TR(IN := wire#w2, R := wire#w3, PV := #V_TOut_TR, BaseUnidades_ms := "CTE_BaseUnidades_1s", QU =>, QD =>, CVU =>, CVD =>)
   END_RUNG
   RUNG wire#powerrail
      Contact( "DB1_SalidasExterioresDeMesa".Mesa[#Mesa].Ir_Pos_E2E4 )
      I_Contact( #Mx_TR_UP_E1E3 )
      wire#w1
      Contact( #EnMovimiento_TRx )
      I_Contact( #EstadoZona.Manual_CBx )
   END_RUNG wire#w2
   RUNG wire#powerrail
      Contact( "DB1_SalidasExterioresDeMesa".Mesa[#Mesa].Ir_Pos_E1E3 )
      Contact( #Mx_TR_UP_E1E3 )
   END_RUNG wire#w1
   RUNG wire#powerrail
      I_Contact( "DB1_SalidasExterioresDeMesa".Mesa[#Mesa].Ir_Pos_E2E4 )
      I_Contact( "DB1_SalidasExterioresDeMesa".Mesa[#Mesa].Ir_Pos_E1E3 )
   END_RUNG wire#w3
   // the same network as SCL:
   #TOut_Subir_TR(IN := (("DB1_SalidasExterioresDeMesa".Mesa[#Mesa].Ir_Pos_E2E4 AND NOT #Mx_TR_UP_E1E3) OR ("DB1_SalidasExterioresDeMesa".Mesa[#Mesa].Ir_Pos_E1E3 AND #Mx_TR_UP_E1E3)) AND #EnMovimiento_TRx AND NOT #EstadoZona.Manual_CBx,   // "FB910_CNT_UHS"
                  R := NOT "DB1_SalidasExterioresDeMesa".Mesa[#Mesa].Ir_Pos_E2E4 AND NOT "DB1_SalidasExterioresDeMesa".Mesa[#Mesa].Ir_Pos_E1E3,
                  PV := #V_TOut_TR,
                  BaseUnidades_ms := "CTE_BaseUnidades_1s");
END_REGION

REGION Network 35: ERROR - Tout Subir TR
   RUNG wire#powerrail
      Contact( #EstadoZona.Rearme_CBx )
      S_RS(operand := #EstadoVI.Err_TOut_Subida, s1 := #TOut_Subir_TR.QU)
      S_Coil( #EstadoVI.Error_Mx )
   END_RUNG
   // the same network as SCL:
   IF #EstadoZona.Rearme_CBx THEN
       #EstadoVI.Err_TOut_Subida := FALSE;   // RS flip-flop
   END_IF;
   IF #TOut_Subir_TR.QU THEN #EstadoVI.Err_TOut_Subida := TRUE; END_IF;
   IF #EstadoVI.Err_TOut_Subida THEN #EstadoVI.Error_Mx := TRUE; END_IF;
END_REGION

REGION Network 36: TMP - ERROR - Tout Bajar Transfer
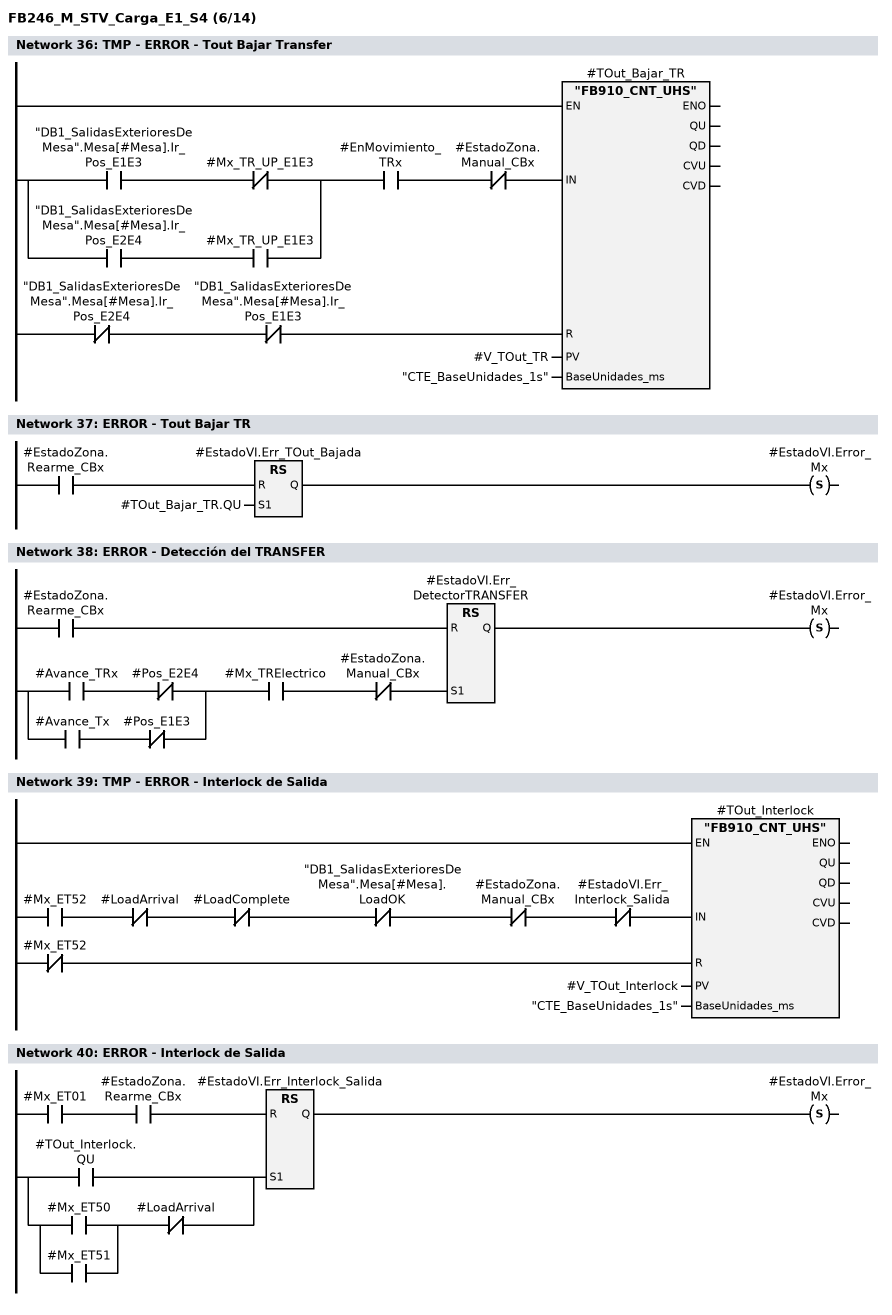
   RUNG wire#powerrail
      #TOut_Bajar_TR(IN := wire#w2, R := wire#w3, PV := #V_TOut_TR, BaseUnidades_ms := "CTE_BaseUnidades_1s", QU =>, QD =>, CVU =>, CVD =>)
   END_RUNG
   RUNG wire#powerrail
      Contact( "DB1_SalidasExterioresDeMesa".Mesa[#Mesa].Ir_Pos_E1E3 )
      I_Contact( #Mx_TR_UP_E1E3 )
      wire#w1
      Contact( #EnMovimiento_TRx )
      I_Contact( #EstadoZona.Manual_CBx )
   END_RUNG wire#w2
   RUNG wire#powerrail
      Contact( "DB1_SalidasExterioresDeMesa".Mesa[#Mesa].Ir_Pos_E2E4 )
      Contact( #Mx_TR_UP_E1E3 )
   END_RUNG wire#w1
   RUNG wire#powerrail
      I_Contact( "DB1_SalidasExterioresDeMesa".Mesa[#Mesa].Ir_Pos_E2E4 )
      I_Contact( "DB1_SalidasExterioresDeMesa".Mesa[#Mesa].Ir_Pos_E1E3 )
   END_RUNG wire#w3
   // the same network as SCL:
   #TOut_Bajar_TR(IN := (("DB1_SalidasExterioresDeMesa".Mesa[#Mesa].Ir_Pos_E1E3 AND NOT #Mx_TR_UP_E1E3) OR ("DB1_SalidasExterioresDeMesa".Mesa[#Mesa].Ir_Pos_E2E4 AND #Mx_TR_UP_E1E3)) AND #EnMovimiento_TRx AND NOT #EstadoZona.Manual_CBx,   // "FB910_CNT_UHS"
                  R := NOT "DB1_SalidasExterioresDeMesa".Mesa[#Mesa].Ir_Pos_E2E4 AND NOT "DB1_SalidasExterioresDeMesa".Mesa[#Mesa].Ir_Pos_E1E3,
                  PV := #V_TOut_TR,
                  BaseUnidades_ms := "CTE_BaseUnidades_1s");
END_REGION

REGION Network 37: ERROR - Tout Bajar TR
   RUNG wire#powerrail
      Contact( #EstadoZona.Rearme_CBx )
      S_RS(operand := #EstadoVI.Err_TOut_Bajada, s1 := #TOut_Bajar_TR.QU)
      S_Coil( #EstadoVI.Error_Mx )
   END_RUNG
   // the same network as SCL:
   IF #EstadoZona.Rearme_CBx THEN
       #EstadoVI.Err_TOut_Bajada := FALSE;   // RS flip-flop
   END_IF;
   IF #TOut_Bajar_TR.QU THEN #EstadoVI.Err_TOut_Bajada := TRUE; END_IF;
   IF #EstadoVI.Err_TOut_Bajada THEN #EstadoVI.Error_Mx := TRUE; END_IF;
END_REGION

REGION Network 38: ERROR - Detección del TRANSFER
   RUNG wire#powerrail
      Contact( #EstadoZona.Rearme_CBx )
      S_RS(operand := #EstadoVI.Err_DetectorTRANSFER, s1 := wire#w2)
      S_Coil( #EstadoVI.Error_Mx )
   END_RUNG
   RUNG wire#powerrail
      Contact( #Avance_TRx )
      I_Contact( #Pos_E2E4 )
      wire#w1
      Contact( #Mx_TRElectrico )
      I_Contact( #EstadoZona.Manual_CBx )
   END_RUNG wire#w2
   RUNG wire#powerrail
      Contact( #Avance_Tx )
      I_Contact( #Pos_E1E3 )
   END_RUNG wire#w1
   // the same network as SCL:
   IF #EstadoZona.Rearme_CBx THEN
       #EstadoVI.Err_DetectorTRANSFER := FALSE;   // RS flip-flop
   END_IF;
   IF ((#Avance_TRx AND NOT #Pos_E2E4) OR (#Avance_Tx AND NOT #Pos_E1E3)) AND #Mx_TRElectrico AND NOT #EstadoZona.Manual_CBx THEN
       #EstadoVI.Err_DetectorTRANSFER := TRUE;
   END_IF;
   IF #EstadoVI.Err_DetectorTRANSFER THEN #EstadoVI.Error_Mx := TRUE; END_IF;
END_REGION

REGION Network 39: TMP - ERROR - Interlock de Salida
   RUNG wire#powerrail
      #TOut_Interlock(IN := wire#w1, R := wire#w2, PV := #V_TOut_Interlock, BaseUnidades_ms := "CTE_BaseUnidades_1s", QU =>, QD =>, CVU =>, CVD =>)
   END_RUNG
   RUNG wire#powerrail
      Contact( #Mx_ET52 )
      I_Contact( #LoadArrival )
      I_Contact( #LoadComplete )
      I_Contact( "DB1_SalidasExterioresDeMesa".Mesa[#Mesa].LoadOK )
      I_Contact( #EstadoZona.Manual_CBx )
      I_Contact( #EstadoVI.Err_Interlock_Salida )
   END_RUNG wire#w1
   RUNG wire#powerrail
      I_Contact( #Mx_ET52 )
   END_RUNG wire#w2
   // the same network as SCL:
   #TOut_Interlock(IN := #Mx_ET52 AND NOT #LoadArrival AND NOT #LoadComplete AND NOT "DB1_SalidasExterioresDeMesa".Mesa[#Mesa].LoadOK AND NOT #EstadoZona.Manual_CBx AND NOT #EstadoVI.Err_Interlock_Salida,   // "FB910_CNT_UHS"
                   R := NOT #Mx_ET52,
                   PV := #V_TOut_Interlock,
                   BaseUnidades_ms := "CTE_BaseUnidades_1s");
END_REGION

REGION Network 40: ERROR - Interlock de Salida
   RUNG wire#powerrail
      Contact( #Mx_ET01 )
      Contact( #EstadoZona.Rearme_CBx )
      S_RS(operand := #EstadoVI.Err_Interlock_Salida, s1 := wire#w2)
      S_Coil( #EstadoVI.Error_Mx )
   END_RUNG
   RUNG wire#powerrail
      Contact( #TOut_Interlock.QU )
   END_RUNG wire#w2
   RUNG wire#powerrail
      Contact( #Mx_ET50 )
      wire#w1
      I_Contact( #LoadArrival )
   END_RUNG wire#w2
   RUNG wire#powerrail
      Contact( #Mx_ET51 )
   END_RUNG wire#w1
   // the same network as SCL:
   IF #Mx_ET01 AND #EstadoZona.Rearme_CBx THEN
       #EstadoVI.Err_Interlock_Salida := FALSE;   // RS flip-flop
   END_IF;
   IF #TOut_Interlock.QU OR ((#Mx_ET50 OR #Mx_ET51) AND NOT #LoadArrival) THEN
       #EstadoVI.Err_Interlock_Salida := TRUE;
   END_IF;
   IF #EstadoVI.Err_Interlock_Salida THEN #EstadoVI.Error_Mx := TRUE; END_IF;
END_REGION

REGION Network 41: CONTROL DE TIEMPO - ERROR - Protrusión (Nota: limitacion de Valor a 1 Segundo)
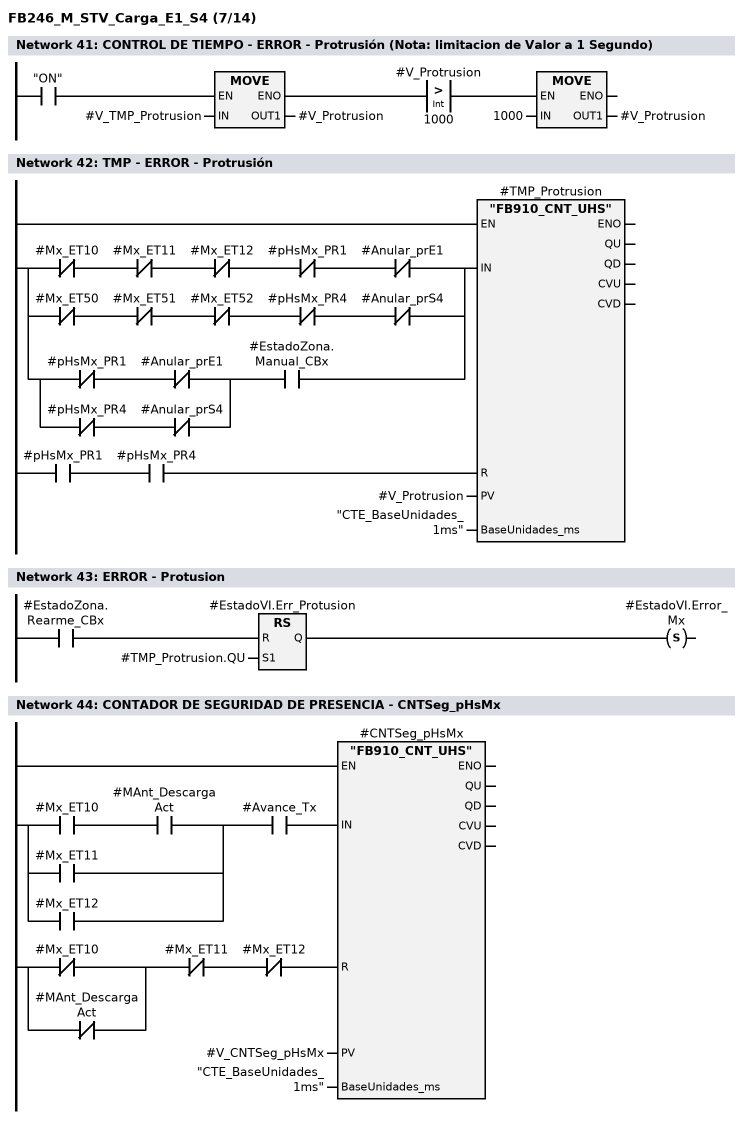
   RUNG wire#powerrail
      Contact( "ON" )
      Move(in := #V_TMP_Protrusion, out1 => #V_Protrusion)
      { S7_Templates := "SrcType := Int" } GT_Contact(in1 := #V_Protrusion, in2 := 1000)
      Move(in := 1000, out1 => #V_Protrusion)
   END_RUNG
   // the same network as SCL:
   IF "ON" THEN #V_Protrusion := #V_TMP_Protrusion; END_IF;
   IF "ON" AND (#V_Protrusion > 1000) THEN #V_Protrusion := 1000; END_IF;
END_REGION

REGION Network 42: TMP - ERROR - Protrusión
   RUNG wire#powerrail
      #TMP_Protrusion(IN := wire#w2, R := wire#w3, PV := #V_Protrusion, BaseUnidades_ms := "CTE_BaseUnidades_1ms", QU =>, QD =>, CVU =>, CVD =>)
   END_RUNG
   RUNG wire#powerrail
      I_Contact( #Mx_ET10 )
      I_Contact( #Mx_ET11 )
      I_Contact( #Mx_ET12 )
      I_Contact( #pHsMx_PR1 )
      I_Contact( #Anular_prE1 )
   END_RUNG wire#w2
   RUNG wire#powerrail
      I_Contact( #Mx_ET50 )
      I_Contact( #Mx_ET51 )
      I_Contact( #Mx_ET52 )
      I_Contact( #pHsMx_PR4 )
      I_Contact( #Anular_prS4 )
   END_RUNG wire#w2
   RUNG wire#powerrail
      I_Contact( #pHsMx_PR1 )
      I_Contact( #Anular_prE1 )
      wire#w1
      Contact( #EstadoZona.Manual_CBx )
   END_RUNG wire#w2
   RUNG wire#powerrail
      I_Contact( #pHsMx_PR4 )
      I_Contact( #Anular_prS4 )
   END_RUNG wire#w1
   RUNG wire#powerrail
      Contact( #pHsMx_PR1 )
      Contact( #pHsMx_PR4 )
   END_RUNG wire#w3
   // the same network as SCL:
   #TMP_Protrusion(IN := (NOT #Mx_ET10 AND NOT #Mx_ET11 AND NOT #Mx_ET12 AND NOT #pHsMx_PR1 AND NOT #Anular_prE1) OR (NOT #Mx_ET50 AND NOT #Mx_ET51 AND NOT #Mx_ET52 AND NOT #pHsMx_PR4 AND NOT #Anular_prS4) OR (((NOT #pHsMx_PR1 AND NOT #Anular_prE1) OR (NOT #pHsMx_PR4 AND NOT #Anular_prS4)) AND #EstadoZona.Manual_CBx),   // "FB910_CNT_UHS"
                   R := #pHsMx_PR1 AND #pHsMx_PR4,
                   PV := #V_Protrusion,
                   BaseUnidades_ms := "CTE_BaseUnidades_1ms");
END_REGION

REGION Network 43: ERROR - Protusion
   RUNG wire#powerrail
      Contact( #EstadoZona.Rearme_CBx )
      S_RS(operand := #EstadoVI.Err_Protusion, s1 := #TMP_Protrusion.QU)
      S_Coil( #EstadoVI.Error_Mx )
   END_RUNG
   // the same network as SCL:
   IF #EstadoZona.Rearme_CBx THEN
       #EstadoVI.Err_Protusion := FALSE;   // RS flip-flop
   END_IF;
   IF #TMP_Protrusion.QU THEN #EstadoVI.Err_Protusion := TRUE; END_IF;
   IF #EstadoVI.Err_Protusion THEN #EstadoVI.Error_Mx := TRUE; END_IF;
END_REGION

REGION Network 44: CONTADOR DE SEGURIDAD DE PRESENCIA - CNTSeg_pHsMx
   RUNG wire#powerrail
      #CNTSeg_pHsMx(IN := wire#w2, R := wire#w4, PV := #V_CNTSeg_pHsMx, BaseUnidades_ms := "CTE_BaseUnidades_1ms", QU =>, QD =>, CVU =>, CVD =>)
   END_RUNG
   RUNG wire#powerrail
      Contact( #Mx_ET10 )
      Contact( #MAnt_DescargaAct )
      wire#w1
      Contact( #Avance_Tx )
   END_RUNG wire#w2
   RUNG wire#powerrail
      Contact( #Mx_ET11 )
   END_RUNG wire#w1
   RUNG wire#powerrail
      Contact( #Mx_ET12 )
   END_RUNG wire#w1
   RUNG wire#powerrail
      I_Contact( #Mx_ET10 )
      wire#w3
      I_Contact( #Mx_ET11 )
      I_Contact( #Mx_ET12 )
   END_RUNG wire#w4
   RUNG wire#powerrail
      I_Contact( #MAnt_DescargaAct )
   END_RUNG wire#w3
   // the same network as SCL:
   #CNTSeg_pHsMx(IN := ((#Mx_ET10 AND #MAnt_DescargaAct) OR #Mx_ET11 OR #Mx_ET12) AND #Avance_Tx,   // "FB910_CNT_UHS"
                 R := (NOT #Mx_ET10 OR NOT #MAnt_DescargaAct) AND NOT #Mx_ET11 AND NOT #Mx_ET12,
                 PV := #V_CNTSeg_pHsMx,
                 BaseUnidades_ms := "CTE_BaseUnidades_1ms");
END_REGION

REGION Network 45: CONTADOR DE PRESENCIA - CNT_pHsMx
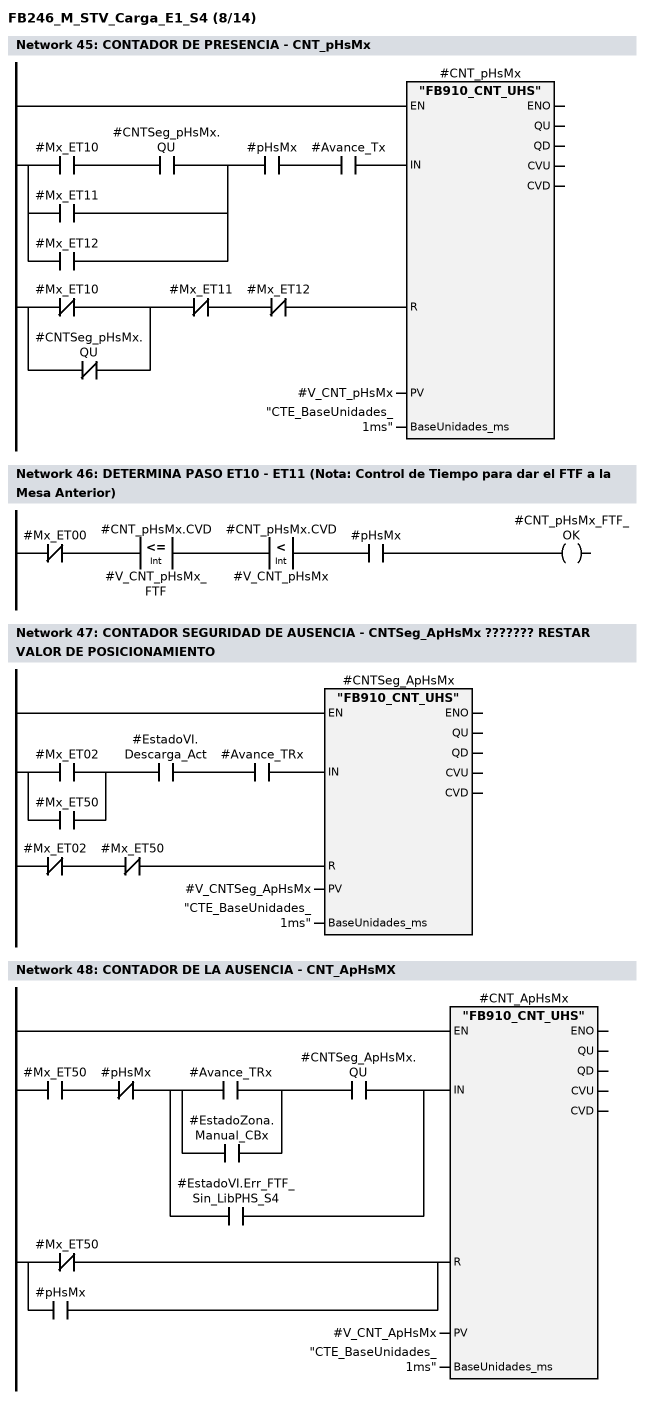
   RUNG wire#powerrail
      #CNT_pHsMx(IN := wire#w2, R := wire#w4, PV := #V_CNT_pHsMx, BaseUnidades_ms := "CTE_BaseUnidades_1ms", QU =>, QD =>, CVU =>, CVD =>)
   END_RUNG
   RUNG wire#powerrail
      Contact( #Mx_ET10 )
      Contact( #CNTSeg_pHsMx.QU )
      wire#w1
      Contact( #pHsMx )
      Contact( #Avance_Tx )
   END_RUNG wire#w2
   RUNG wire#powerrail
      Contact( #Mx_ET11 )
   END_RUNG wire#w1
   RUNG wire#powerrail
      Contact( #Mx_ET12 )
   END_RUNG wire#w1
   RUNG wire#powerrail
      I_Contact( #Mx_ET10 )
      wire#w3
      I_Contact( #Mx_ET11 )
      I_Contact( #Mx_ET12 )
   END_RUNG wire#w4
   RUNG wire#powerrail
      I_Contact( #CNTSeg_pHsMx.QU )
   END_RUNG wire#w3
   // the same network as SCL:
   #CNT_pHsMx(IN := ((#Mx_ET10 AND #CNTSeg_pHsMx.QU) OR #Mx_ET11 OR #Mx_ET12) AND #pHsMx AND #Avance_Tx,   // "FB910_CNT_UHS"
              R := (NOT #Mx_ET10 OR NOT #CNTSeg_pHsMx.QU) AND NOT #Mx_ET11 AND NOT #Mx_ET12,
              PV := #V_CNT_pHsMx,
              BaseUnidades_ms := "CTE_BaseUnidades_1ms");
END_REGION

REGION Network 46: DETERMINA PASO ET10 - ET11 (Nota: Control de Tiempo para dar el FTF a la Mesa Anterior)
   RUNG wire#powerrail
      I_Contact( #Mx_ET00 )
      { S7_Templates := "SrcType := Int" } LE_Contact(in1 := #CNT_pHsMx.CVD, in2 := #V_CNT_pHsMx_FTF)
      { S7_Templates := "SrcType := Int" } LT_Contact(in1 := #CNT_pHsMx.CVD, in2 := #V_CNT_pHsMx)
      Contact( #pHsMx )
      Coil( #CNT_pHsMx_FTF_OK )
   END_RUNG
   // the same network as SCL:
   #CNT_pHsMx_FTF_OK := NOT #Mx_ET00 AND (#CNT_pHsMx.CVD <= #V_CNT_pHsMx_FTF) AND (#CNT_pHsMx.CVD < #V_CNT_pHsMx) AND #pHsMx;
END_REGION

REGION Network 47: CONTADOR SEGURIDAD DE AUSENCIA - CNTSeg_ApHsMx ??????? RESTAR VALOR DE POSICIONAMIENTO
   RUNG wire#powerrail
      #CNTSeg_ApHsMx(IN := wire#w2, R := wire#w3, PV := #V_CNTSeg_ApHsMx, BaseUnidades_ms := "CTE_BaseUnidades_1ms", QU =>, QD =>, CVU =>, CVD =>)
   END_RUNG
   RUNG wire#powerrail
      Contact( #Mx_ET02 )
      wire#w1
      Contact( #EstadoVI.Descarga_Act )
      Contact( #Avance_TRx )
   END_RUNG wire#w2
   RUNG wire#powerrail
      Contact( #Mx_ET50 )
   END_RUNG wire#w1
   RUNG wire#powerrail
      I_Contact( #Mx_ET02 )
      I_Contact( #Mx_ET50 )
   END_RUNG wire#w3
   // the same network as SCL:
   #CNTSeg_ApHsMx(IN := (#Mx_ET02 OR #Mx_ET50) AND #EstadoVI.Descarga_Act AND #Avance_TRx,   // "FB910_CNT_UHS"
                  R := NOT #Mx_ET02 AND NOT #Mx_ET50,
                  PV := #V_CNTSeg_ApHsMx,
                  BaseUnidades_ms := "CTE_BaseUnidades_1ms");
END_REGION

REGION Network 48: CONTADOR DE LA AUSENCIA - CNT_ApHsMX
   RUNG wire#powerrail
      #CNT_ApHsMx(IN := wire#w3, R := wire#w4, PV := #V_CNT_ApHsMx, BaseUnidades_ms := "CTE_BaseUnidades_1ms", QU =>, QD =>, CVU =>, CVD =>)
   END_RUNG
   RUNG wire#powerrail
      Contact( #Mx_ET50 )
      I_Contact( #pHsMx )
      wire#w1
      Contact( #Avance_TRx )
      wire#w2
      Contact( #CNTSeg_ApHsMx.QU )
   END_RUNG wire#w3
   RUNG wire#w1
      Contact( #EstadoZona.Manual_CBx )
   END_RUNG wire#w2
   RUNG wire#w1
      Contact( #EstadoVI.Err_FTF_Sin_LibPHS_S4 )
   END_RUNG wire#w3
   RUNG wire#powerrail
      I_Contact( #Mx_ET50 )
   END_RUNG wire#w4
   RUNG wire#powerrail
      Contact( #pHsMx )
   END_RUNG wire#w4
   // the same network as SCL:
   #CNT_ApHsMx(IN := #Mx_ET50 AND NOT #pHsMx AND (((#Avance_TRx OR #EstadoZona.Manual_CBx) AND #CNTSeg_ApHsMx.QU) OR #EstadoVI.Err_FTF_Sin_LibPHS_S4),   // "FB910_CNT_UHS"
               R := NOT #Mx_ET50 OR #pHsMx,
               PV := #V_CNT_ApHsMx,
               BaseUnidades_ms := "CTE_BaseUnidades_1ms");
END_REGION

REGION Network 49: VARIABLES AUXILIARES - Fin de Reset
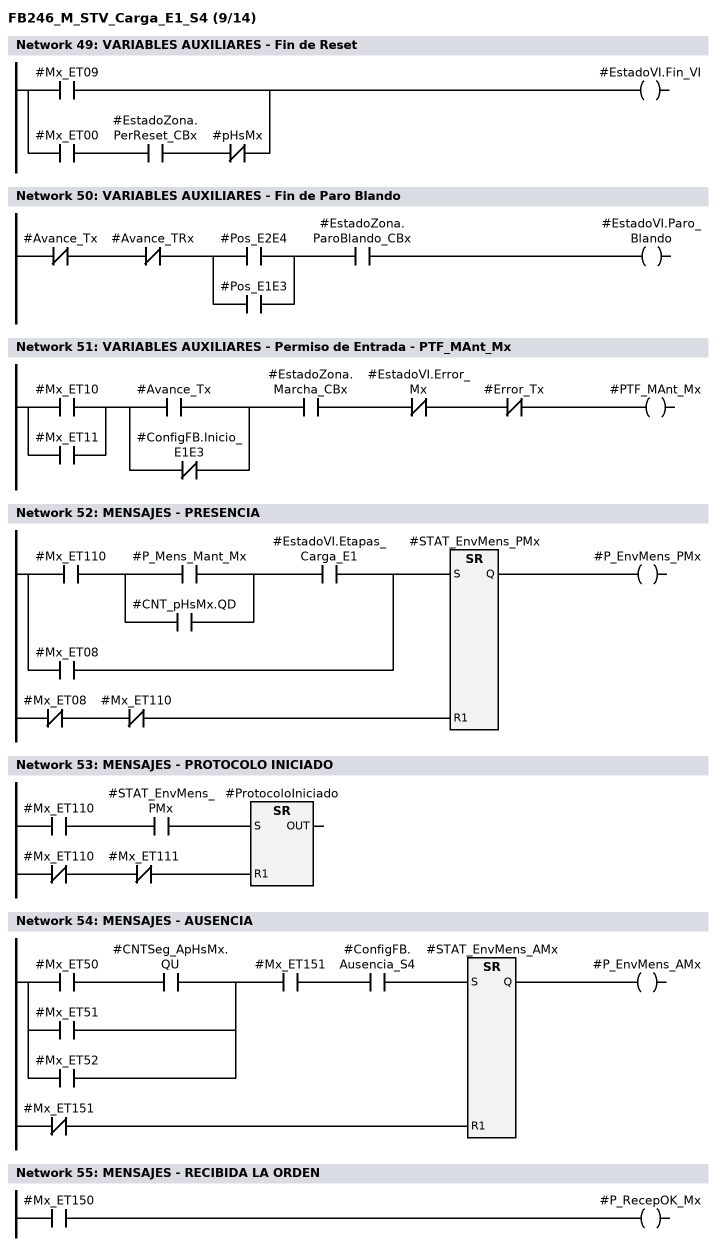
   RUNG wire#powerrail
      Contact( #Mx_ET09 )
      wire#w1
      Coil( #EstadoVI.Fin_VI )
   END_RUNG
   RUNG wire#powerrail
      Contact( #Mx_ET00 )
      Contact( #EstadoZona.PerReset_CBx )
      I_Contact( #pHsMx )
   END_RUNG wire#w1
   // the same network as SCL:
   #EstadoVI.Fin_VI := #Mx_ET09 OR (#Mx_ET00 AND #EstadoZona.PerReset_CBx AND NOT #pHsMx);
END_REGION

REGION Network 50: VARIABLES AUXILIARES - Fin de Paro Blando
   RUNG wire#powerrail
      I_Contact( #Avance_Tx )
      I_Contact( #Avance_TRx )
      wire#w1
      Contact( #Pos_E2E4 )
      wire#w2
      Contact( #EstadoZona.ParoBlando_CBx )
      Coil( #EstadoVI.Paro_Blando )
   END_RUNG
   RUNG wire#w1
      Contact( #Pos_E1E3 )
   END_RUNG wire#w2
   // the same network as SCL:
   #EstadoVI.Paro_Blando := NOT #Avance_Tx AND NOT #Avance_TRx AND (#Pos_E2E4 OR #Pos_E1E3) AND #EstadoZona.ParoBlando_CBx;
END_REGION

REGION Network 51: VARIABLES AUXILIARES - Permiso de Entrada - PTF_MAnt_Mx
   RUNG wire#powerrail
      Contact( #Mx_ET10 )
      wire#w1
      Contact( #Avance_Tx )
      wire#w2
      Contact( #EstadoZona.Marcha_CBx )
      I_Contact( #EstadoVI.Error_Mx )
      I_Contact( #Error_Tx )
      Coil( #PTF_MAnt_Mx )
   END_RUNG
   RUNG wire#powerrail
      Contact( #Mx_ET11 )
   END_RUNG wire#w1
   RUNG wire#w1
      I_Contact( #ConfigFB.Inicio_E1E3 )
   END_RUNG wire#w2
   // the same network as SCL:
   #PTF_MAnt_Mx := (#Mx_ET10 OR #Mx_ET11) AND (#Avance_Tx OR NOT #ConfigFB.Inicio_E1E3) AND #EstadoZona.Marcha_CBx AND NOT #EstadoVI.Error_Mx AND NOT #Error_Tx;
END_REGION

REGION Network 52: MENSAJES - PRESENCIA
   RUNG wire#powerrail
      Contact( #Mx_ET110 )
      wire#w1
      Contact( #P_Mens_Mant_Mx )
      wire#w2
      Contact( #EstadoVI.Etapas_Carga_E1 )
      wire#w3
      S_SR(operand := #STAT_EnvMens_PMx, r1 := wire#w4)
      Coil( #P_EnvMens_PMx )
   END_RUNG
   RUNG wire#w1
      Contact( #CNT_pHsMx.QD )
   END_RUNG wire#w2
   RUNG wire#powerrail
      Contact( #Mx_ET08 )
   END_RUNG wire#w3
   RUNG wire#powerrail
      I_Contact( #Mx_ET08 )
      I_Contact( #Mx_ET110 )
   END_RUNG wire#w4
   // the same network as SCL:
   IF (#Mx_ET110 AND (#P_Mens_Mant_Mx OR #CNT_pHsMx.QD) AND #EstadoVI.Etapas_Carga_E1) OR #Mx_ET08 THEN
       #STAT_EnvMens_PMx := TRUE;   // SR flip-flop
   END_IF;
   IF NOT #Mx_ET08 AND NOT #Mx_ET110 THEN #STAT_EnvMens_PMx := FALSE; END_IF;
   #P_EnvMens_PMx := #STAT_EnvMens_PMx;
END_REGION

REGION Network 53: MENSAJES - PROTOCOLO INICIADO
   RUNG wire#powerrail
      Contact( #Mx_ET110 )
      Contact( #STAT_EnvMens_PMx )
      S_SR(operand := #ProtocoloIniciado, r1 := wire#w1)
   END_RUNG
   RUNG wire#powerrail
      I_Contact( #Mx_ET110 )
      I_Contact( #Mx_ET111 )
   END_RUNG wire#w1
   // the same network as SCL:
   IF #Mx_ET110 AND #STAT_EnvMens_PMx THEN
       #ProtocoloIniciado := TRUE;   // SR flip-flop
   END_IF;
   IF NOT #Mx_ET110 AND NOT #Mx_ET111 THEN #ProtocoloIniciado := FALSE; END_IF;
END_REGION

REGION Network 54: MENSAJES - AUSENCIA
   RUNG wire#powerrail
      Contact( #Mx_ET50 )
      Contact( #CNTSeg_ApHsMx.QU )
      wire#w1
      Contact( #Mx_ET151 )
      Contact( #ConfigFB.Ausencia_S4 )
      S_SR(operand := #STAT_EnvMens_AMx, r1 := wire#w2)
      Coil( #P_EnvMens_AMx )
   END_RUNG
   RUNG wire#powerrail
      Contact( #Mx_ET51 )
   END_RUNG wire#w1
   RUNG wire#powerrail
      Contact( #Mx_ET52 )
   END_RUNG wire#w1
   RUNG wire#powerrail
      I_Contact( #Mx_ET151 )
   END_RUNG wire#w2
   // the same network as SCL:
   IF ((#Mx_ET50 AND #CNTSeg_ApHsMx.QU) OR #Mx_ET51 OR #Mx_ET52) AND #Mx_ET151 AND #ConfigFB.Ausencia_S4 THEN
       #STAT_EnvMens_AMx := TRUE;   // SR flip-flop
   END_IF;
   IF NOT #Mx_ET151 THEN #STAT_EnvMens_AMx := FALSE; END_IF;
   #P_EnvMens_AMx := #STAT_EnvMens_AMx;
END_REGION

REGION Network 55: MENSAJES - RECIBIDA LA ORDEN
   RUNG wire#powerrail
      Contact( #Mx_ET150 )
      Coil( #P_RecepOK_Mx )
   END_RUNG
   // the same network as SCL:
   #P_RecepOK_Mx := #Mx_ET150;
END_REGION

REGION Network 56: SALIDAS - Interlock de Carga al VTD - LOAD_OK
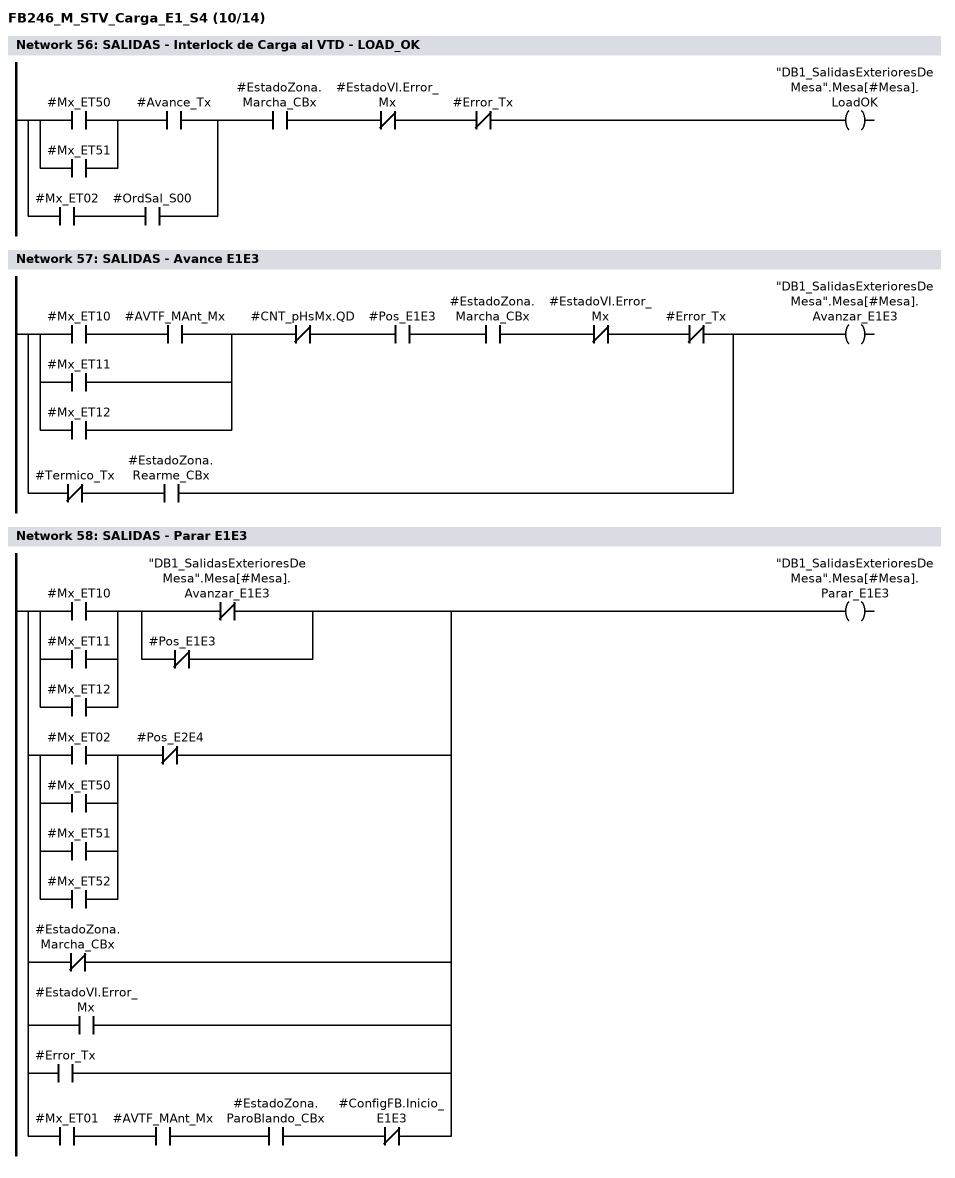
   RUNG wire#powerrail
      Contact( #Mx_ET50 )
      wire#w1
      Contact( #Avance_Tx )
      wire#w2
      Contact( #EstadoZona.Marcha_CBx )
      I_Contact( #EstadoVI.Error_Mx )
      I_Contact( #Error_Tx )
      Coil( "DB1_SalidasExterioresDeMesa".Mesa[#Mesa].LoadOK )
   END_RUNG
   RUNG wire#powerrail
      Contact( #Mx_ET51 )
   END_RUNG wire#w1
   RUNG wire#powerrail
      Contact( #Mx_ET02 )
      Contact( #OrdSal_S00 )
   END_RUNG wire#w2
   // the same network as SCL:
   "DB1_SalidasExterioresDeMesa".Mesa[#Mesa].LoadOK := (((#Mx_ET50 OR #Mx_ET51) AND #Avance_Tx) OR (#Mx_ET02 AND #OrdSal_S00)) AND #EstadoZona.Marcha_CBx AND NOT #EstadoVI.Error_Mx AND NOT #Error_Tx;
END_REGION

REGION Network 57: SALIDAS - Avance E1E3
   RUNG wire#powerrail
      Contact( #Mx_ET10 )
      Contact( #AVTF_MAnt_Mx )
      wire#w1
      I_Contact( #CNT_pHsMx.QD )
      Contact( #Pos_E1E3 )
      Contact( #EstadoZona.Marcha_CBx )
      I_Contact( #EstadoVI.Error_Mx )
      I_Contact( #Error_Tx )
      wire#w2
      Coil( "DB1_SalidasExterioresDeMesa".Mesa[#Mesa].Avanzar_E1E3 )
   END_RUNG
   RUNG wire#powerrail
      Contact( #Mx_ET11 )
   END_RUNG wire#w1
   RUNG wire#powerrail
      Contact( #Mx_ET12 )
   END_RUNG wire#w1
   RUNG wire#powerrail
      I_Contact( #Termico_Tx )
      Contact( #EstadoZona.Rearme_CBx )
   END_RUNG wire#w2
   // the same network as SCL:
   "DB1_SalidasExterioresDeMesa".Mesa[#Mesa].Avanzar_E1E3 := (((#Mx_ET10 AND #AVTF_MAnt_Mx) OR #Mx_ET11 OR #Mx_ET12) AND NOT #CNT_pHsMx.QD AND #Pos_E1E3 AND #EstadoZona.Marcha_CBx AND NOT #EstadoVI.Error_Mx AND NOT #Error_Tx) OR (NOT #Termico_Tx AND #EstadoZona.Rearme_CBx);
END_REGION

REGION Network 58: SALIDAS - Parar E1E3
   RUNG wire#powerrail
      Contact( #Mx_ET10 )
      wire#w1
      I_Contact( "DB1_SalidasExterioresDeMesa".Mesa[#Mesa].Avanzar_E1E3 )
      wire#w2
      Coil( "DB1_SalidasExterioresDeMesa".Mesa[#Mesa].Parar_E1E3 )
   END_RUNG
   RUNG wire#powerrail
      Contact( #Mx_ET11 )
   END_RUNG wire#w1
   RUNG wire#powerrail
      Contact( #Mx_ET12 )
   END_RUNG wire#w1
   RUNG wire#w1
      I_Contact( #Pos_E1E3 )
   END_RUNG wire#w2
   RUNG wire#powerrail
      Contact( #Mx_ET02 )
      wire#w3
      I_Contact( #Pos_E2E4 )
   END_RUNG wire#w2
   RUNG wire#powerrail
      Contact( #Mx_ET50 )
   END_RUNG wire#w3
   RUNG wire#powerrail
      Contact( #Mx_ET51 )
   END_RUNG wire#w3
   RUNG wire#powerrail
      Contact( #Mx_ET52 )
   END_RUNG wire#w3
   RUNG wire#powerrail
      I_Contact( #EstadoZona.Marcha_CBx )
   END_RUNG wire#w2
   RUNG wire#powerrail
      Contact( #EstadoVI.Error_Mx )
   END_RUNG wire#w2
   RUNG wire#powerrail
      Contact( #Error_Tx )
   END_RUNG wire#w2
   RUNG wire#powerrail
      Contact( #Mx_ET01 )
      Contact( #AVTF_MAnt_Mx )
      Contact( #EstadoZona.ParoBlando_CBx )
      I_Contact( #ConfigFB.Inicio_E1E3 )
   END_RUNG wire#w2
   // the same network as SCL:
   "DB1_SalidasExterioresDeMesa".Mesa[#Mesa].Parar_E1E3 := ((#Mx_ET10 OR #Mx_ET11 OR #Mx_ET12) AND (NOT "DB1_SalidasExterioresDeMesa".Mesa[#Mesa].Avanzar_E1E3 OR NOT #Pos_E1E3)) OR ((#Mx_ET02 OR #Mx_ET50 OR #Mx_ET51 OR #Mx_ET52) AND NOT #Pos_E2E4) OR NOT #EstadoZona.Marcha_CBx OR #EstadoVI.Error_Mx OR #Error_Tx OR (#Mx_ET01 AND #AVTF_MAnt_Mx AND #EstadoZona.ParoBlando_CBx AND NOT #ConfigFB.Inicio_E1E3);
END_REGION

REGION Network 59: SALIDAS - Valor Frecuencia Lenta E1E3
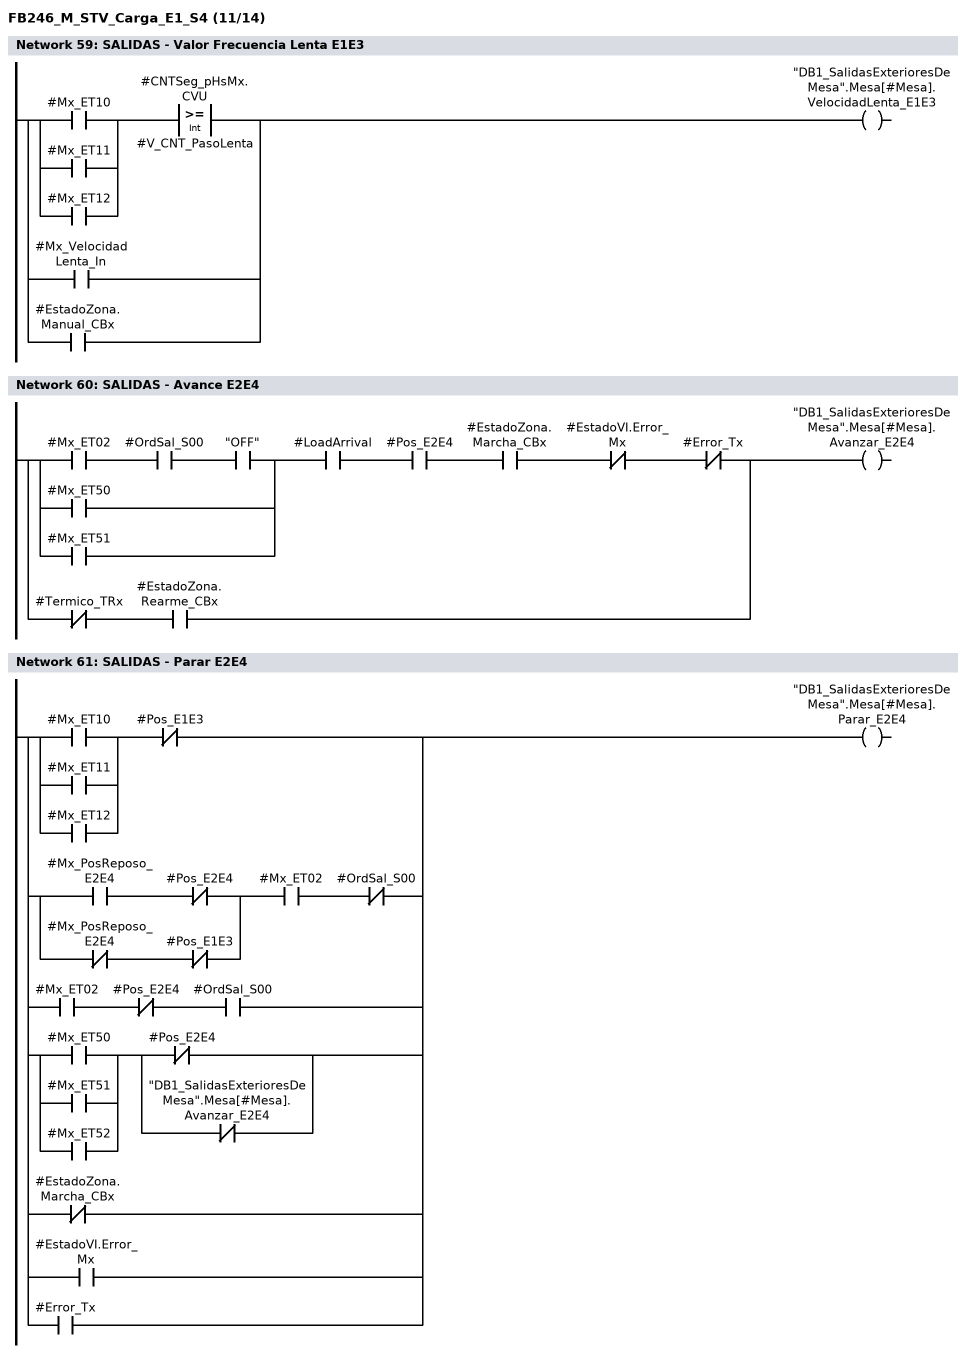
   RUNG wire#powerrail
      Contact( #Mx_ET10 )
      wire#w1
      { S7_Templates := "SrcType := Int" } GE_Contact(in1 := #CNTSeg_pHsMx.CVU, in2 := #V_CNT_PasoLenta)
      wire#w2
      Coil( "DB1_SalidasExterioresDeMesa".Mesa[#Mesa].VelocidadLenta_E1E3 )
   END_RUNG
   RUNG wire#powerrail
      Contact( #Mx_ET11 )
   END_RUNG wire#w1
   RUNG wire#powerrail
      Contact( #Mx_ET12 )
   END_RUNG wire#w1
   RUNG wire#powerrail
      Contact( #Mx_VelocidadLenta_In )
   END_RUNG wire#w2
   RUNG wire#powerrail
      Contact( #EstadoZona.Manual_CBx )
   END_RUNG wire#w2
   // the same network as SCL:
   "DB1_SalidasExterioresDeMesa".Mesa[#Mesa].VelocidadLenta_E1E3 := ((#Mx_ET10 OR #Mx_ET11 OR #Mx_ET12) AND (#CNTSeg_pHsMx.CVU >= #V_CNT_PasoLenta)) OR #Mx_VelocidadLenta_In OR #EstadoZona.Manual_CBx;
END_REGION

REGION Network 60: SALIDAS - Avance E2E4
   RUNG wire#powerrail
      Contact( #Mx_ET02 )
      Contact( #OrdSal_S00 )
      Contact( "OFF" )
      wire#w1
      Contact( #LoadArrival )
      Contact( #Pos_E2E4 )
      Contact( #EstadoZona.Marcha_CBx )
      I_Contact( #EstadoVI.Error_Mx )
      I_Contact( #Error_Tx )
      wire#w2
      Coil( "DB1_SalidasExterioresDeMesa".Mesa[#Mesa].Avanzar_E2E4 )
   END_RUNG
   RUNG wire#powerrail
      Contact( #Mx_ET50 )
   END_RUNG wire#w1
   RUNG wire#powerrail
      Contact( #Mx_ET51 )
   END_RUNG wire#w1
   RUNG wire#powerrail
      I_Contact( #Termico_TRx )
      Contact( #EstadoZona.Rearme_CBx )
   END_RUNG wire#w2
   // the same network as SCL:
   "DB1_SalidasExterioresDeMesa".Mesa[#Mesa].Avanzar_E2E4 := (((#Mx_ET02 AND #OrdSal_S00 AND "OFF") OR #Mx_ET50 OR #Mx_ET51) AND #LoadArrival AND #Pos_E2E4 AND #EstadoZona.Marcha_CBx AND NOT #EstadoVI.Error_Mx AND NOT #Error_Tx) OR (NOT #Termico_TRx AND #EstadoZona.Rearme_CBx);
END_REGION

REGION Network 61: SALIDAS - Parar E2E4
   RUNG wire#powerrail
      Contact( #Mx_ET10 )
      wire#w1
      I_Contact( #Pos_E1E3 )
      wire#w2
      Coil( "DB1_SalidasExterioresDeMesa".Mesa[#Mesa].Parar_E2E4 )
   END_RUNG
   RUNG wire#powerrail
      Contact( #Mx_ET11 )
   END_RUNG wire#w1
   RUNG wire#powerrail
      Contact( #Mx_ET12 )
   END_RUNG wire#w1
   RUNG wire#powerrail
      Contact( #Mx_PosReposo_E2E4 )
      I_Contact( #Pos_E2E4 )
      wire#w3
      Contact( #Mx_ET02 )
      I_Contact( #OrdSal_S00 )
   END_RUNG wire#w2
   RUNG wire#powerrail
      I_Contact( #Mx_PosReposo_E2E4 )
      I_Contact( #Pos_E1E3 )
   END_RUNG wire#w3
   RUNG wire#powerrail
      Contact( #Mx_ET02 )
      I_Contact( #Pos_E2E4 )
      Contact( #OrdSal_S00 )
   END_RUNG wire#w2
   RUNG wire#powerrail
      Contact( #Mx_ET50 )
      wire#w4
      I_Contact( #Pos_E2E4 )
   END_RUNG wire#w2
   RUNG wire#powerrail
      Contact( #Mx_ET51 )
   END_RUNG wire#w4
   RUNG wire#powerrail
      Contact( #Mx_ET52 )
   END_RUNG wire#w4
   RUNG wire#w4
      I_Contact( "DB1_SalidasExterioresDeMesa".Mesa[#Mesa].Avanzar_E2E4 )
   END_RUNG wire#w2
   RUNG wire#powerrail
      I_Contact( #EstadoZona.Marcha_CBx )
   END_RUNG wire#w2
   RUNG wire#powerrail
      Contact( #EstadoVI.Error_Mx )
   END_RUNG wire#w2
   RUNG wire#powerrail
      Contact( #Error_Tx )
   END_RUNG wire#w2
   // the same network as SCL:
   "DB1_SalidasExterioresDeMesa".Mesa[#Mesa].Parar_E2E4 := ((#Mx_ET10 OR #Mx_ET11 OR #Mx_ET12) AND NOT #Pos_E1E3) OR (((#Mx_PosReposo_E2E4 AND NOT #Pos_E2E4) OR (NOT #Mx_PosReposo_E2E4 AND NOT #Pos_E1E3)) AND #Mx_ET02 AND NOT #OrdSal_S00) OR (#Mx_ET02 AND NOT #Pos_E2E4 AND #OrdSal_S00) OR ((#Mx_ET50 OR #Mx_ET51 OR #Mx_ET52) AND (NOT #Pos_E2E4 OR NOT "DB1_SalidasExterioresDeMesa".Mesa[#Mesa].Avanzar_E2E4)) OR NOT #EstadoZona.Marcha_CBx OR #EstadoVI.Error_Mx OR #Error_Tx;
END_REGION

REGION Network 62: SALIDAS - Valor Frecuencia Lenta E2E4
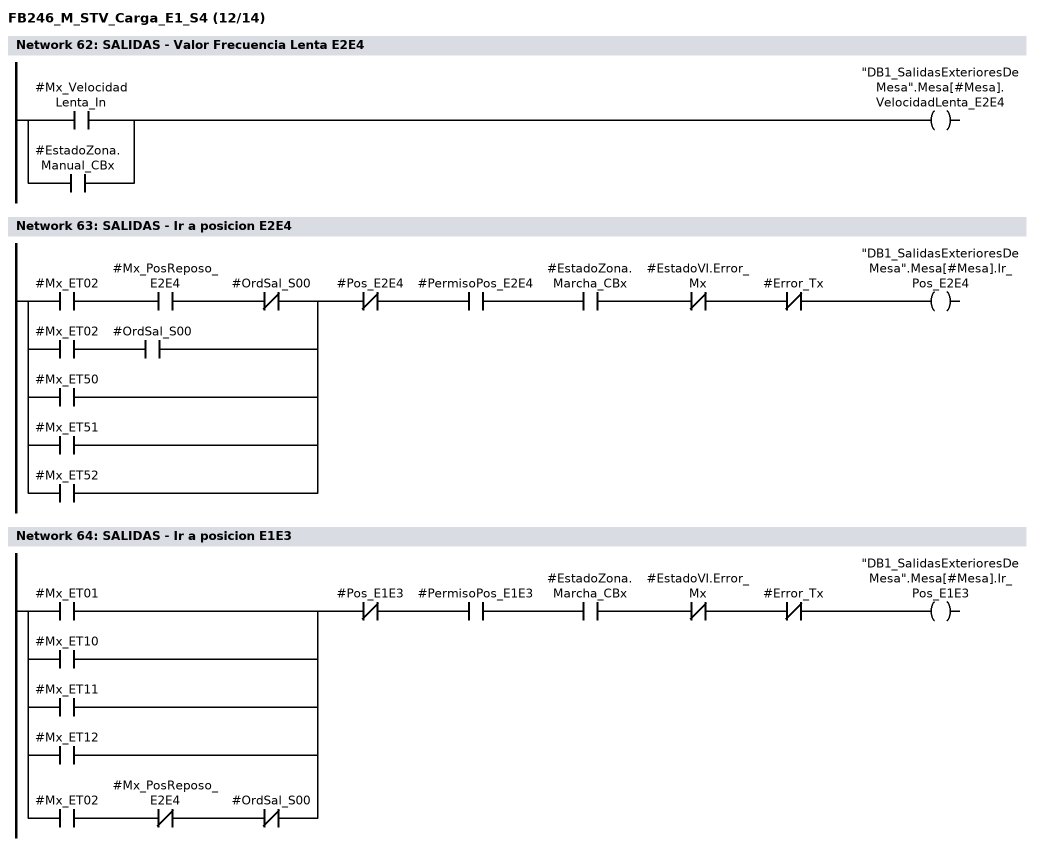
   RUNG wire#powerrail
      Contact( #Mx_VelocidadLenta_In )
      wire#w1
      Coil( "DB1_SalidasExterioresDeMesa".Mesa[#Mesa].VelocidadLenta_E2E4 )
   END_RUNG
   RUNG wire#powerrail
      Contact( #EstadoZona.Manual_CBx )
   END_RUNG wire#w1
   // the same network as SCL:
   "DB1_SalidasExterioresDeMesa".Mesa[#Mesa].VelocidadLenta_E2E4 := #Mx_VelocidadLenta_In OR #EstadoZona.Manual_CBx;
END_REGION

REGION Network 63: SALIDAS - Ir a posicion E2E4
   RUNG wire#powerrail
      Contact( #Mx_ET02 )
      Contact( #Mx_PosReposo_E2E4 )
      I_Contact( #OrdSal_S00 )
      wire#w1
      I_Contact( #Pos_E2E4 )
      Contact( #PermisoPos_E2E4 )
      Contact( #EstadoZona.Marcha_CBx )
      I_Contact( #EstadoVI.Error_Mx )
      I_Contact( #Error_Tx )
      Coil( "DB1_SalidasExterioresDeMesa".Mesa[#Mesa].Ir_Pos_E2E4 )
   END_RUNG
   RUNG wire#powerrail
      Contact( #Mx_ET02 )
      Contact( #OrdSal_S00 )
   END_RUNG wire#w1
   RUNG wire#powerrail
      Contact( #Mx_ET50 )
   END_RUNG wire#w1
   RUNG wire#powerrail
      Contact( #Mx_ET51 )
   END_RUNG wire#w1
   RUNG wire#powerrail
      Contact( #Mx_ET52 )
   END_RUNG wire#w1
   // the same network as SCL:
   "DB1_SalidasExterioresDeMesa".Mesa[#Mesa].Ir_Pos_E2E4 := ((#Mx_ET02 AND #Mx_PosReposo_E2E4 AND NOT #OrdSal_S00) OR (#Mx_ET02 AND #OrdSal_S00) OR #Mx_ET50 OR #Mx_ET51 OR #Mx_ET52) AND NOT #Pos_E2E4 AND #PermisoPos_E2E4 AND #EstadoZona.Marcha_CBx AND NOT #EstadoVI.Error_Mx AND NOT #Error_Tx;
END_REGION

REGION Network 64: SALIDAS - Ir a posicion E1E3
   RUNG wire#powerrail
      Contact( #Mx_ET01 )
      wire#w1
      I_Contact( #Pos_E1E3 )
      Contact( #PermisoPos_E1E3 )
      Contact( #EstadoZona.Marcha_CBx )
      I_Contact( #EstadoVI.Error_Mx )
      I_Contact( #Error_Tx )
      Coil( "DB1_SalidasExterioresDeMesa".Mesa[#Mesa].Ir_Pos_E1E3 )
   END_RUNG
   RUNG wire#powerrail
      Contact( #Mx_ET10 )
   END_RUNG wire#w1
   RUNG wire#powerrail
      Contact( #Mx_ET11 )
   END_RUNG wire#w1
   RUNG wire#powerrail
      Contact( #Mx_ET12 )
   END_RUNG wire#w1
   RUNG wire#powerrail
      Contact( #Mx_ET02 )
      I_Contact( #Mx_PosReposo_E2E4 )
      I_Contact( #OrdSal_S00 )
   END_RUNG wire#w1
   // the same network as SCL:
   "DB1_SalidasExterioresDeMesa".Mesa[#Mesa].Ir_Pos_E1E3 := (#Mx_ET01 OR #Mx_ET10 OR #Mx_ET11 OR #Mx_ET12 OR (#Mx_ET02 AND NOT #Mx_PosReposo_E2E4 AND NOT #OrdSal_S00)) AND NOT #Pos_E1E3 AND #PermisoPos_E1E3 AND #EstadoZona.Marcha_CBx AND NOT #EstadoVI.Error_Mx AND NOT #Error_Tx;
END_REGION

REGION Network 65: ESTADOS DE LA MESA
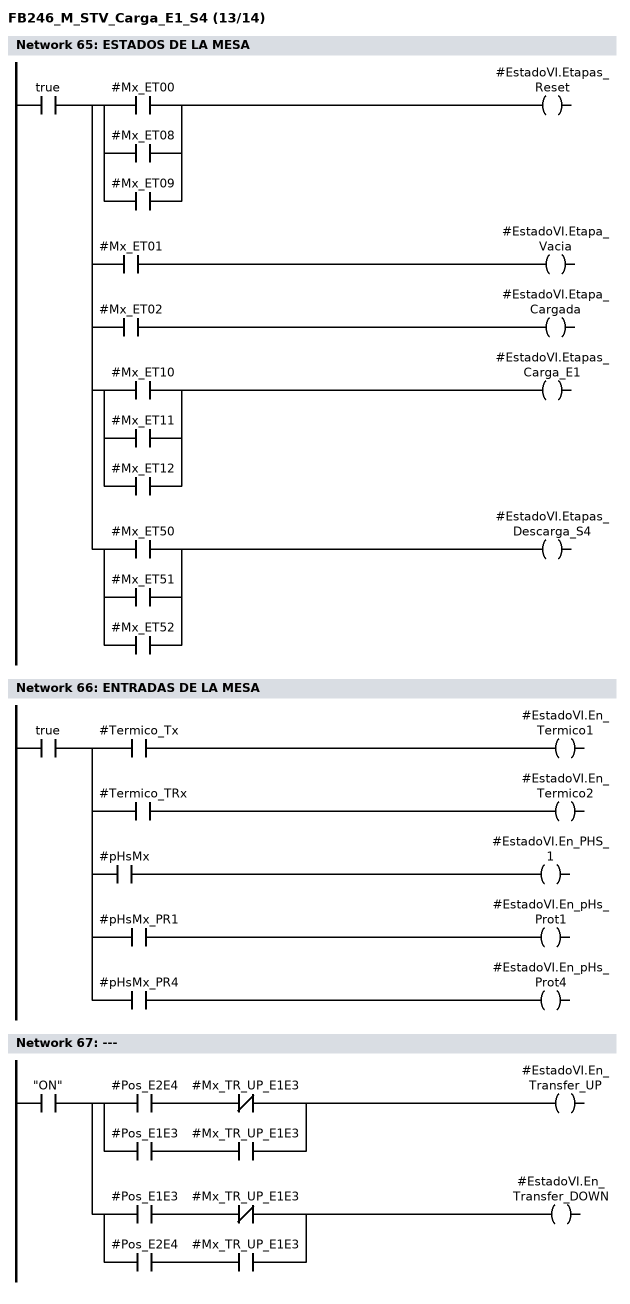
   RUNG wire#powerrail
      Contact( true )
      wire#w1
      Contact( #Mx_ET00 )
      wire#w2
      Coil( #EstadoVI.Etapas_Reset )
   END_RUNG
   RUNG wire#w1
      Contact( #Mx_ET08 )
   END_RUNG wire#w2
   RUNG wire#w1
      Contact( #Mx_ET09 )
   END_RUNG wire#w2
   RUNG wire#w1
      Contact( #Mx_ET01 )
      Coil( #EstadoVI.Etapa_Vacia )
   END_RUNG
   RUNG wire#w1
      Contact( #Mx_ET02 )
      Coil( #EstadoVI.Etapa_Cargada )
   END_RUNG
   RUNG wire#w1
      Contact( #Mx_ET10 )
      wire#w3
      Coil( #EstadoVI.Etapas_Carga_E1 )
   END_RUNG
   RUNG wire#w1
      Contact( #Mx_ET11 )
   END_RUNG wire#w3
   RUNG wire#w1
      Contact( #Mx_ET12 )
   END_RUNG wire#w3
   RUNG wire#w1
      Contact( #Mx_ET50 )
      wire#w4
      Coil( #EstadoVI.Etapas_Descarga_S4 )
   END_RUNG
   RUNG wire#w1
      Contact( #Mx_ET51 )
   END_RUNG wire#w4
   RUNG wire#w1
      Contact( #Mx_ET52 )
   END_RUNG wire#w4
   // the same network as SCL:
   #EstadoVI.Etapas_Reset := true AND (#Mx_ET00 OR #Mx_ET08 OR #Mx_ET09);
   #EstadoVI.Etapa_Vacia := true AND #Mx_ET01;
   #EstadoVI.Etapa_Cargada := true AND #Mx_ET02;
   #EstadoVI.Etapas_Carga_E1 := true AND (#Mx_ET10 OR #Mx_ET11 OR #Mx_ET12);
   #EstadoVI.Etapas_Descarga_S4 := true AND (#Mx_ET50 OR #Mx_ET51 OR #Mx_ET52);
END_REGION

REGION Network 66: ENTRADAS DE LA MESA
   RUNG wire#powerrail
      Contact( true )
      wire#w1
      Contact( #Termico_Tx )
      Coil( #EstadoVI.En_Termico1 )
   END_RUNG
   RUNG wire#w1
      Contact( #Termico_TRx )
      Coil( #EstadoVI.En_Termico2 )
   END_RUNG
   RUNG wire#w1
      Contact( #pHsMx )
      Coil( #EstadoVI.En_PHS_1 )
   END_RUNG
   RUNG wire#w1
      Contact( #pHsMx_PR1 )
      Coil( #EstadoVI.En_pHs_Prot1 )
   END_RUNG
   RUNG wire#w1
      Contact( #pHsMx_PR4 )
      Coil( #EstadoVI.En_pHs_Prot4 )
   END_RUNG
   // the same network as SCL:
   #EstadoVI.En_Termico1 := true AND #Termico_Tx;
   #EstadoVI.En_Termico2 := true AND #Termico_TRx;
   #EstadoVI.En_PHS_1 := true AND #pHsMx;
   #EstadoVI.En_pHs_Prot1 := true AND #pHsMx_PR1;
   #EstadoVI.En_pHs_Prot4 := true AND #pHsMx_PR4;
END_REGION

REGION Network 67: ---
   RUNG wire#powerrail
      Contact( "ON" )
      wire#w1
      Contact( #Pos_E2E4 )
      I_Contact( #Mx_TR_UP_E1E3 )
      wire#w2
      Coil( #EstadoVI.En_Transfer_UP )
   END_RUNG
   RUNG wire#w1
      Contact( #Pos_E1E3 )
      Contact( #Mx_TR_UP_E1E3 )
   END_RUNG wire#w2
   RUNG wire#w1
      Contact( #Pos_E1E3 )
      I_Contact( #Mx_TR_UP_E1E3 )
      wire#w3
      Coil( #EstadoVI.En_Transfer_DOWN )
   END_RUNG
   RUNG wire#w1
      Contact( #Pos_E2E4 )
      Contact( #Mx_TR_UP_E1E3 )
   END_RUNG wire#w3
   // the same network as SCL:
   #EstadoVI.En_Transfer_UP := "ON" AND ((#Pos_E2E4 AND NOT #Mx_TR_UP_E1E3) OR (#Pos_E1E3 AND #Mx_TR_UP_E1E3));
   #EstadoVI.En_Transfer_DOWN := "ON" AND ((#Pos_E1E3 AND NOT #Mx_TR_UP_E1E3) OR (#Pos_E2E4 AND #Mx_TR_UP_E1E3));
END_REGION

REGION Network 68: SALIDAS DE LA MESA
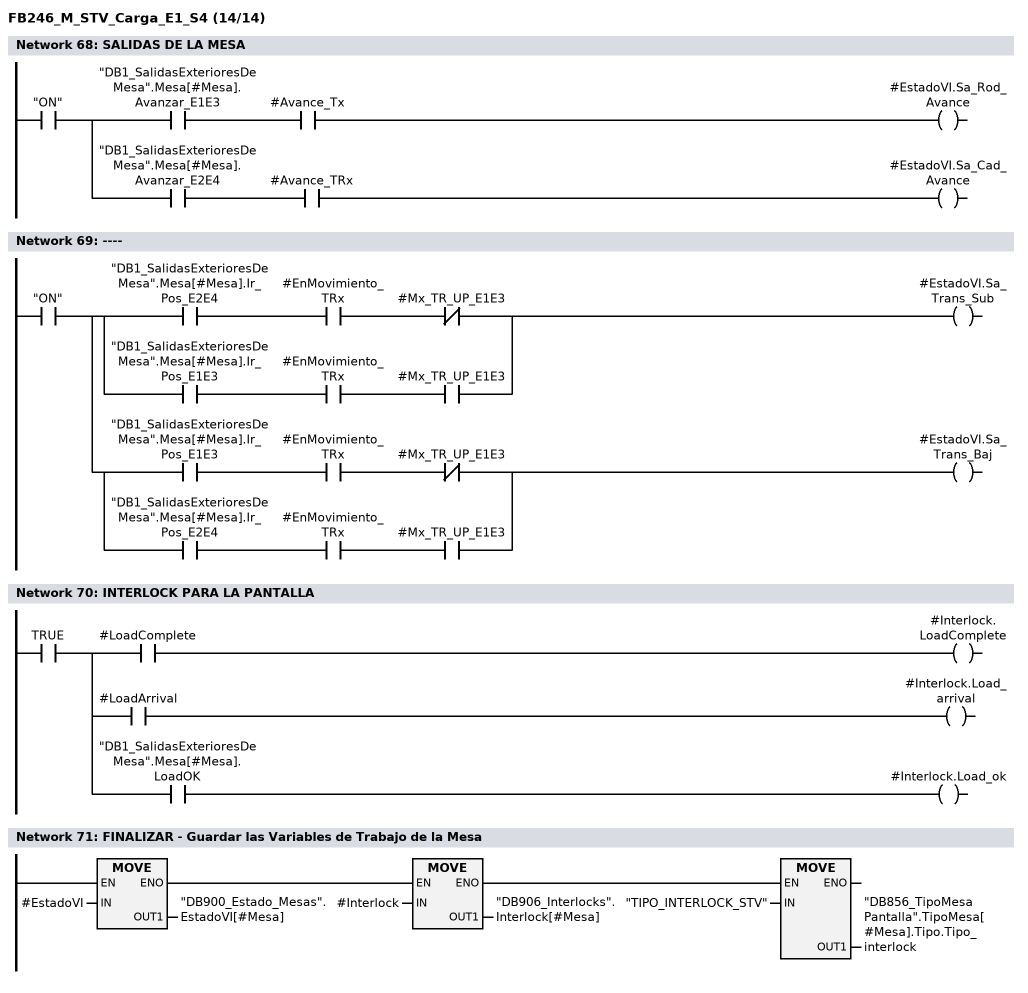
   RUNG wire#powerrail
      Contact( "ON" )
      wire#w1
      Contact( "DB1_SalidasExterioresDeMesa".Mesa[#Mesa].Avanzar_E1E3 )
      Contact( #Avance_Tx )
      Coil( #EstadoVI.Sa_Rod_Avance )
   END_RUNG
   RUNG wire#w1
      Contact( "DB1_SalidasExterioresDeMesa".Mesa[#Mesa].Avanzar_E2E4 )
      Contact( #Avance_TRx )
      Coil( #EstadoVI.Sa_Cad_Avance )
   END_RUNG
   // the same network as SCL:
   #EstadoVI.Sa_Rod_Avance := "ON" AND "DB1_SalidasExterioresDeMesa".Mesa[#Mesa].Avanzar_E1E3 AND #Avance_Tx;
   #EstadoVI.Sa_Cad_Avance := "ON" AND "DB1_SalidasExterioresDeMesa".Mesa[#Mesa].Avanzar_E2E4 AND #Avance_TRx;
END_REGION

REGION Network 69: ----
   RUNG wire#powerrail
      Contact( "ON" )
      wire#w1
      Contact( "DB1_SalidasExterioresDeMesa".Mesa[#Mesa].Ir_Pos_E2E4 )
      Contact( #EnMovimiento_TRx )
      I_Contact( #Mx_TR_UP_E1E3 )
      wire#w2
      Coil( #EstadoVI.Sa_Trans_Sub )
   END_RUNG
   RUNG wire#w1
      Contact( "DB1_SalidasExterioresDeMesa".Mesa[#Mesa].Ir_Pos_E1E3 )
      Contact( #EnMovimiento_TRx )
      Contact( #Mx_TR_UP_E1E3 )
   END_RUNG wire#w2
   RUNG wire#w1
      Contact( "DB1_SalidasExterioresDeMesa".Mesa[#Mesa].Ir_Pos_E1E3 )
      Contact( #EnMovimiento_TRx )
      I_Contact( #Mx_TR_UP_E1E3 )
      wire#w3
      Coil( #EstadoVI.Sa_Trans_Baj )
   END_RUNG
   RUNG wire#w1
      Contact( "DB1_SalidasExterioresDeMesa".Mesa[#Mesa].Ir_Pos_E2E4 )
      Contact( #EnMovimiento_TRx )
      Contact( #Mx_TR_UP_E1E3 )
   END_RUNG wire#w3
   // the same network as SCL:
   #EstadoVI.Sa_Trans_Sub := "ON" AND (("DB1_SalidasExterioresDeMesa".Mesa[#Mesa].Ir_Pos_E2E4 AND #EnMovimiento_TRx AND NOT #Mx_TR_UP_E1E3) OR ("DB1_SalidasExterioresDeMesa".Mesa[#Mesa].Ir_Pos_E1E3 AND #EnMovimiento_TRx AND #Mx_TR_UP_E1E3));
   #EstadoVI.Sa_Trans_Baj := "ON" AND (("DB1_SalidasExterioresDeMesa".Mesa[#Mesa].Ir_Pos_E1E3 AND #EnMovimiento_TRx AND NOT #Mx_TR_UP_E1E3) OR ("DB1_SalidasExterioresDeMesa".Mesa[#Mesa].Ir_Pos_E2E4 AND #EnMovimiento_TRx AND #Mx_TR_UP_E1E3));
END_REGION

REGION Network 70: INTERLOCK PARA LA PANTALLA
   RUNG wire#powerrail
      Contact( TRUE )
      wire#w1
      Contact( #LoadComplete )
      Coil( #Interlock.LoadComplete )
   END_RUNG
   RUNG wire#w1
      Contact( #LoadArrival )
      Coil( #Interlock.Load_arrival )
   END_RUNG
   RUNG wire#w1
      Contact( "DB1_SalidasExterioresDeMesa".Mesa[#Mesa].LoadOK )
      Coil( #Interlock.Load_ok )
   END_RUNG
   // the same network as SCL:
   #Interlock.LoadComplete := TRUE AND #LoadComplete;
   #Interlock.Load_arrival := TRUE AND #LoadArrival;
   #Interlock.Load_ok := TRUE AND "DB1_SalidasExterioresDeMesa".Mesa[#Mesa].LoadOK;
END_REGION

REGION Network 71: FINALIZAR - Guardar las Variables de Trabajo de la Mesa
   RUNG wire#powerrail
      Move(in := #EstadoVI, out1 => "DB900_Estado_Mesas".EstadoVI[#Mesa])
      Move(in := #Interlock, out1 => "DB906_Interlocks".Interlock[#Mesa])
      Move(in := "TIPO_INTERLOCK_STV", out1 => "DB856_TipoMesaPantalla".TipoMesa[#Mesa].Tipo.Tipo_interlock)
   END_RUNG
   // the same network as SCL:
   "DB900_Estado_Mesas".EstadoVI[#Mesa] := #EstadoVI;
   "DB906_Interlocks".Interlock[#Mesa] := #Interlock;
   "DB856_TipoMesaPantalla".TipoMesa[#Mesa].Tipo.Tipo_interlock := "TIPO_INTERLOCK_STV";
END_REGION
END_FUNCTION_BLOCK
